(* Logix 5000 project; controller P3 vendor 1 type 14 code 92 rev 20.55; software revision 20.01 *)

TASK MainTask (continuous, watchdog 500 ms) : MainProgram

MODULES
   Local : vendor 1 type 14 code 92 (ICP 0, rev 20.55)
      P3_EN2T_PCN : 1756-EN2T (ICP 1, Ethernet 192.168.1.30, rev 10.1)
         P2 : 1756-EN2T (Ethernet 192.168.1.20, rev 10.1, Output RPI 10 ms)
            P2_CONTROLLER : vendor 1 type 14 code 92 (ICP 0, rev 20.1)
         P4 : 1756-EN2T (Ethernet 192.168.1.40, rev 10.1, Output RPI 10 ms)
            P4_CONTROLLER : vendor 1 type 14 code 92 (ICP 0, rev 20.1)
         P6 : 1756-EN2T (Ethernet 192.168.1.60, rev 10.1, Output RPI 10 ms)
            P6_CONTROLLER : vendor 1 type 14 code 92 (ICP 0, rev 20.1)
         EN2T_P1 : 1756-EN2T (Ethernet 192.168.1.10, rev 10.1, Output RPI 10 ms)
            P1_CONTROLLER : vendor 1 type 14 code 92 (ICP 0, rev 20.1)
         P5 : 1756-EN2T (Ethernet 192.168.1.50, rev 10.7, Output RPI 10 ms)
            P5_CONTROLLER : vendor 1 type 14 code 92 (ICP 0, rev 20.55)
      P3_EN2TR_RIO : vendor 1 type 12 code 200 (ICP 2, Ethernet 192.168.0.30, rev 10.1)
         RIO3 : 1794-AENTR (Ethernet 192.168.0.32, rev 1.1, Output RPI 20 ms)
            RIO3_DI : 1794-IB32 (Flex 0, rev 1.1, Input RPI 20 ms)
            RIO3_DO : vendor 1 type 7 code 35 (Flex 1, rev 1.1)
            RIO3_AI : 1794-IE12 (Flex 2, rev 1.1, Output RPI 78 ms)
         WRIO3 : vendor 309 type 12 code 1000 (Ethernet 192.168.0.35, rev 3.1, Output RPI 20 ms)
            WRIO3_AI : 1734-IE4C (PointIO 1, rev 3.1, Input RPI 80 ms)
END_MODULES

TYPE AIN_UDT :
STRUCT
   Pv : REAL;
   Heu : REAL;
   Leu : REAL;
   SAHH : REAL;
   SAH : REAL;
   SAL : REAL;
   SALL : REAL;
   AHH : BOOL;
   AH : BOOL;
   AL : BOOL;
   ALL : BOOL;
   Wifi_Enb : BOOL;
   Hty : BOOL;
   Sim : BOOL;
   Sim_PV : REAL;
END_STRUCT
END_TYPE

TYPE AUTOINP_UDT :
STRUCT
   ON : BOOL;
END_STRUCT
END_TYPE

TYPE ControllerLEDStatus :
STRUCT
   Off : BOOL;
   SolidGreen : BOOL;
   FlashingGreen : BOOL;
   SolidYellow : BOOL;
   FlashingYellow : BOOL;
   FlashingRed : BOOL;
   SolidRed : BOOL;
END_STRUCT
END_TYPE

TYPE Duty2_UDT :
STRUCT
   Selection : INT;
   Pump_Running : BOOL;
   Selected_Pmp_Not_Avl : BOOL;
   Both_Pmp_Not_Avl : BOOL;
END_STRUCT
END_TYPE

TYPE FaultRecord :
STRUCT
   timelow : DINT;
   timehigh : DINT;
   type : INT;
   code : INT;
   info : DINT[8];
END_STRUCT
END_TYPE

TYPE FIT_UDT :
STRUCT
   Pv : REAL;
   Heu : REAL;
   Leu : REAL;
   SAHH : REAL;
   SAH : REAL;
   SAL : REAL;
   SALL : REAL;
   Totaliser : REAL;
   AHH : BOOL;
   AH : BOOL;
   AL : BOOL;
   ALL : BOOL;
   Sim : BOOL;
   Sim_PV : REAL;
   Wifi_Enb : BOOL;
   Rst_Totaliser : BOOL;
   Hty : BOOL;
END_STRUCT
END_TYPE

TYPE Logix_Status_FP :
STRUCT
   ClearMinorFaults : DINT;
   Sts_MinorFaultEvents : DINT;
   Sts_MinorFaultBits : DINT;
   Sts_Redundant : DINT;
   Set_FaceplateAnimation : DINT;
   Val_ProductCode : DINT;
   MemoryTemp : INT[29];
   Val_raw_data : INT;
   Sts_IO_LED_raw : INT;
   Sts_ProductCode : INT;
   Val_Force_data_raw : INT;
   MemoryRequestData : SINT[12];
   Sts_Force_Installed : BOOL;
   Sts_Force_Enabled : BOOL;
   Sts_Faulted : BOOL;
   Sts_Run : BOOL;
   Sts_Program : BOOL;
   Sts_Minor_fault : BOOL;
   Sts_Major_fault : BOOL;
   Sts_KS_in_run : BOOL;
   Sts_KS_in_program : BOOL;
   Sts_KS_in_remote : BOOL;
   Sts_Changingmodes : BOOL;
   Sts_Test : BOOL;
   Sts_Ladder_Working : BOOL;
   Cmd_ClearFaultRecord : BOOL;
   Set_Controller_Description : STRING;
   UpdateDelayTimer : TIMER;
   Val_MajorFault : FaultRecord;
   Val_MFS : FaultRecord;
   Sts_IO_LED : ControllerLEDStatus;
   Sts_Battery_LED : ControllerLEDStatus;
   MemoryData : Memory_Data;
   TEST : DINT;
END_STRUCT
END_TYPE

TYPE Memory_Data :
STRUCT
   Free_Mem_IO : DINT;
   Free_Mem_DT : DINT;
   Free_Memory : DINT;
   Total_Mem_IO : DINT;
   Total_Mem_DT : DINT;
   Total_Memory : DINT;
   Biggest_IO_Mem_Size_Ava : DINT;
   Biggest_DT_Mem_Size_Ava : DINT;
END_STRUCT
END_TYPE

TYPE MV_UDT :
STRUCT
   Cmd : INT;
   Status : INT;
   Reset : BOOL;
   Auto : BOOL;
   FTO : BOOL;
   FTC : BOOL;
   Avl : BOOL;
END_STRUCT
END_TYPE

TYPE PLANT_AUTO_UDT :
STRUCT
   ON : BOOL;
   OFF : BOOL;
END_STRUCT
END_TYPE

TYPE PLANT_UDT :
STRUCT
   START : BOOL;
   STOP : BOOL;
END_STRUCT
END_TYPE

TYPE PMP_UDT :
STRUCT
   Cmd : INT;
   Status : INT;
   RunMin : REAL;
   Total_RunMin : REAL;
   RunHr : REAL;
   Total_RunHr : REAL;
   Remote : BOOL;
   Auto : BOOL;
   Fault : BOOL;
   Avl : BOOL;
   Permissive : DINT;
   Shutdown : DINT;
   SD : DINT;
   Reset : BOOL;
   Reset_RunHr : BOOL;
   FTR : BOOL;
   FTS : BOOL;
END_STRUCT
END_TYPE

TYPE PRECONDITION_UDT :
STRUCT
   PERMISSIVE1 : BOOL;
   PERMISSIVE2 : BOOL;
   PERMISSIVE3 : BOOL;
   PERMISSIVE4 : BOOL;
   PERMISSIVE5 : BOOL;
   SHUTDOWN1 : BOOL;
   SHUTDOWN2 : BOOL;
   SHUTDOWN3 : BOOL;
   SHUTDOWN4 : BOOL;
   SHUTDOWN5 : BOOL;
END_STRUCT
END_TYPE

TYPE RED_STAT :
STRUCT
   Redundancy_status_of_the_controller : INT;
   Redundancy_state_of_the_partner : INT;
END_STRUCT
END_TYPE

TYPE SWITCH_UDT :
STRUCT
   Alarm : BOOL;
   Delay : DINT;
END_STRUCT
END_TYPE

TYPE WIFI_UDT :
STRUCT
   PLC_WIFI : BOOL;
   RIO_WIFI : BOOL;
END_STRUCT
END_TYPE

ADD_ON_INSTRUCTION AIN_FBD   (* revision 1.0 *)
VAR_INPUT
   WRIO_Enb : BOOL; {visible}
   Raw_RIO : INT; {visible}
   Raw_WRIO : INT; {visible}
   L_Raw_RIO : INT; {visible}
   H_Raw_RIO : INT; {visible}
   L_Raw_WRIO : INT; {visible}
   H_Raw_WRIO : INT; {visible}
   HEU : INT; {visible}
   LEU : INT; {visible}
END_VAR
VAR_OUTPUT
   Hty : BOOL; {visible}
   Wifi_Enb : BOOL; {access Read Only, visible}
   AHH : BOOL; {visible}
   AH : BOOL; {access Read Only, visible}
   AL : BOOL; {access Read Only, visible}
   ALL : BOOL; {visible}
END_VAR
VAR_INPUT
   SAHH : REAL; {visible}
   SAH : REAL; {visible}
   SAL : REAL; {visible}
   SALL : REAL; {visible}
   Simulation : BOOL; {visible}
   RIO_Hty : BOOL; {visible}
   WRIO_Hty : BOOL; {visible}
END_VAR
VAR_IN_OUT
   Pv : REAL; {required}
   Sim_PV : REAL; {required}
   HMI : AIN_UDT; {required}
END_VAR
VAR
   SCALE : SCALE; {access None}
   ALM : ALARM; {access None}
   _Raw : INT; {access None}
   _L_Raw : INT; {access None}
   _H_Raw : INT; {access None}
   _Inst_Hty : BOOL; {access None}
END_VAR

ROUTINE Logic   (* structured text *)
   (*RIO and Wireless RIO Selection*)
   
   IF WRIO_Enb THEN
   	Wifi_Enb	:= 1;
   	_Raw		:= Raw_WRIO;
   	_H_Raw		:= H_Raw_WRIO;
   	_L_Raw		:= L_Raw_WRIO;
   	_Inst_Hty 	:= WRIO_Hty;
   ELSE
   	Wifi_Enb	:= 0;
   	_Raw		:= Raw_RIO;
   	_H_Raw		:= H_Raw_RIO;
   	_L_Raw		:= L_Raw_RIO;
   	_Inst_Hty 	:= RIO_Hty;
   END_IF;
   
   (*Calculation for PV*)
   IF Simulation THEN
   	Pv	:=Sim_PV;
   ELSE
   	SCALE.In		:=_Raw;
   	SCALE.InRawMax	:=_H_Raw;
   	SCALE.InRawMin	:=_L_Raw;
   	SCALE.InEUMax	:=HEU;
   	SCALE.InEUMin	:=LEU;
   	SCL(SCALE);
   
   	IF SCALE.Out<0 THEN
   		Pv	:= 0.0;
   	ELSE
   		Pv	:=SCALE.Out;
   	END_IF;
   
   	Sim_PV	:=Pv;
   
   END_IF;
   
   (*Alarms*)
   ALM.In			:=Pv;
   ALM.HHLimit		:=SAHH;
   ALM.HLimit		:=SAH;
   ALM.LLimit		:=SAL;
   ALM.LLLimit		:=SALL;
   ALM(ALM);
   
   AHH				:=ALM.HHAlarm;
   AH				:=ALM.HAlarm;
   AL				:=ALM.LAlarm;
   ALL				:=ALM.LLAlarm;
   
   Hty:= _Inst_Hty AND (_Raw > _L_Raw) AND (_Raw < _H_Raw)  ;
   
   
   
   
   
   
END_ROUTINE
END_ADD_ON_INSTRUCTION

ADD_ON_INSTRUCTION Duty2_FBD   (* revision 1.0 *)
VAR_INPUT
   AutoInp : BOOL; {visible}
   Selection : INT; {visible}
END_VAR
VAR_OUTPUT
   Start_Pmp1 : BOOL; {visible}
   Start_Pmp2 : BOOL; {visible}
END_VAR
VAR_IN_OUT
   PMP1 : PMP_UDT; {required}
   PMP2 : PMP_UDT; {required}
   HMI : Duty2_UDT; {required}
END_VAR

ROUTINE Logic   (* structured text *)
   IF PMP1.Status=2 OR PMP2.Status=2 THEN
   	HMI.Pump_Running := 1;
   ELSE
   	HMI.Pump_Running := 0;
   END_IF;
   
   IF AutoInp THEN
   	CASE Selection OF
   		(*PUMP 1 *)
   		1:
   			IF PMP1.Avl THEN
   				Start_Pmp1					:=1;
   				Start_Pmp2					:=0;
   				HMI.Selected_Pmp_Not_Avl	:=0;
   			ELSIF NOT PMP1.Avl AND PMP2.Avl THEN
   				Start_Pmp1					:=0;
   				Start_Pmp2					:=1;
   				HMI.Selected_Pmp_Not_Avl	:=1;
   			ELSIF NOT PMP1.Avl AND NOT PMP2.Avl	THEN
   				Start_Pmp1					:=0;
   				Start_Pmp2					:=0;
   				HMI.Both_Pmp_Not_Avl		:=1;
   			END_IF;
   
   		(*PUMP 2 *)
   		2:
   			IF PMP2.Avl THEN
   				Start_Pmp1					:=0;
   				Start_Pmp2					:=1;
   				HMI.Selected_Pmp_Not_Avl	:=0;
   			ELSIF NOT PMP2.Avl AND PMP1.Avl THEN
   				Start_Pmp1					:=1;
   				Start_Pmp2					:=0;
   				HMI.Selected_Pmp_Not_Avl	:=1;
   			ELSIF NOT PMP1.Avl AND NOT PMP2.Avl	THEN
   				Start_Pmp1					:=0;
   				Start_Pmp2					:=0;
   				HMI.Both_Pmp_Not_Avl		:=1;
   			END_IF;
   	END_CASE;
   ELSE
   	Start_Pmp1					:=0;
   	Start_Pmp2					:=0;
   END_IF;
   
   
END_ROUTINE
END_ADD_ON_INSTRUCTION

ADD_ON_INSTRUCTION FIT_FBD   (* revision 1.0 *)
VAR_INPUT
   WRIO_Enb : BOOL; {visible}
   Raw_RIO : INT; {visible}
   Raw_WRIO : INT; {visible}
   L_Raw_RIO : INT; {visible}
   H_Raw_RIO : INT; {visible}
   L_Raw_WRIO : INT; {visible}
   H_Raw_WRIO : INT; {visible}
   HEU : REAL; {visible}
   LEU : REAL; {visible}
END_VAR
VAR_OUTPUT
   Hty : BOOL; {visible}
   Wifi_Enb : BOOL; {visible}
   AHH : BOOL; {visible}
   AH : BOOL; {access Read Only, visible}
   AL : BOOL; {access Read Only, visible}
   ALL : BOOL; {visible}
END_VAR
VAR_INPUT
   SAHH : REAL; {visible}
   SAH : REAL; {visible}
   SAL : REAL; {visible}
   SALL : REAL; {visible}
   Simulation : BOOL; {visible}
   RIO_Hty : BOOL; {visible}
   WRIO_Hty : BOOL; {visible}
   Totaliser_Enb : BOOL; {visible}
   Rst_Totaliser : BOOL; {visible}
END_VAR
VAR_IN_OUT
   Totaliser : REAL; {required}
   Pv : REAL; {required}
   Sim_Pv : REAL; {required}
   HMI : FIT_UDT; {required}
END_VAR
VAR
   SCALE : SCALE; {access None}
   ALM : ALARM; {access None}
   TON : FBD_TIMER; {access None}
   _SEC_P : BOOL; {access None}
   _Inst_Hty : BOOL; {access None}
   _L_Raw : INT; {access None}
   _H_Raw : INT; {access None}
   _Raw : INT; {access None}
   R_TRIG : FBD_ONESHOT; {access None}
END_VAR

ROUTINE Logic   (* structured text *)
   (*RIO and Wireless RIO Selection*)
   
   IF WRIO_Enb THEN
   	Wifi_Enb	:= 1;
   	_Raw		:= Raw_WRIO;
   	_H_Raw		:= H_Raw_WRIO;
   	_L_Raw		:= L_Raw_WRIO;
   	_Inst_Hty 	:= WRIO_Hty;
   ELSE
   	Wifi_Enb	:= 0;
   	_Raw		:= Raw_RIO;
   	_H_Raw		:= H_Raw_RIO;
   	_L_Raw		:= L_Raw_RIO;
   	_Inst_Hty 	:= RIO_Hty;
   END_IF;
   
   (*Calculation for PV*)
   IF Simulation THEN
   	Pv	:= Sim_Pv   ;
   ELSE
   	SCALE.In		:=_Raw;
   	SCALE.InRawMax	:=_H_Raw;
   	SCALE.InRawMin	:=_L_Raw;
   	SCALE.InEUMax	:=HEU;
   	SCALE.InEUMin	:=LEU;
   	SCL(SCALE);
   	IF SCALE.Out>0 THEN
   		Pv	:=SCALE.Out;
   	ELSIF SCALE.Out<=0 THEN
   		Pv	:=0.0;
   	END_IF;
   
   	Sim_Pv	:=Pv;
   END_IF;
   
   (*Alarms*)
   ALM.In			:=Pv;
   ALM.HHLimit		:=SAHH;
   ALM.HLimit		:=SAH;
   ALM.LLimit		:=SAL;
   ALM.LLLimit		:=SALL;
   ALM(ALM);
   
   AHH				:=ALM.HHAlarm;
   AH				:=ALM.HAlarm;
   AL				:=ALM.LAlarm;
   ALL				:=ALM.LLAlarm;
   
   (*SECOND PULSE*)
   TON.PRE	:=1000;
   TON.TimerEnable	:=1;
   TONR(TON );
   R_TRIG.InputBit :=TON.DN ;
   OSRI( R_TRIG);
   _SEC_P  := R_TRIG.OutputBit;
   TON.Reset := _SEC_P;
   
   IF Totaliser_Enb THEN
   	IF _SEC_P THEN
   		HMI.Totaliser := HMI.Totaliser +  (ABS(Pv) / 3600 );
   	END_IF;
   END_IF;
   
   IF  Rst_Totaliser   THEN
   	HMI.Totaliser	:=0;
   END_IF;
   
   Hty:= _Inst_Hty AND (_Raw > _L_Raw) AND (_Raw < _H_Raw)  ;
   
   
   
   
   
   
END_ROUTINE
END_ADD_ON_INSTRUCTION

ADD_ON_INSTRUCTION MV_FBD   (* revision 1.0 *)
VAR_INPUT
   Auto : BOOL; {visible}
END_VAR
VAR_OUTPUT
   Cmd_Open : BOOL; {visible}
   Cmd_Close : BOOL; {visible}
   FTO : BOOL; {visible}
   FTC : BOOL; {access Read Only, visible}
END_VAR
VAR_INPUT
   AutoInp : BOOL; {visible}
   ZSO : BOOL; {visible}
   Open_TM : DINT; {visible}
   ZSC : BOOL; {visible}
   Close_TM : DINT; {visible}
END_VAR
VAR_IN_OUT
   Cmd : INT; {required}
   HMI : MV_UDT; {required}
END_VAR
VAR
   TON_Open_TM : FBD_TIMER; {access None}
   TON_Close_TM : FBD_TIMER; {access None}
END_VAR

ROUTINE Logic   (* structured text *)
   (*Fail to Close*)
   TON_Close_TM.PRE 			:= 	Close_TM*1000;
   TON_Close_TM.TimerEnable 	:=  Cmd_Close;
   TONR(TON_Close_TM);
   
   (*Fail to Open*)
   TON_Open_TM.PRE 			:= 	Open_TM*1000;
   TON_Open_TM.TimerEnable 	:= 	Cmd_Open;
   TONR(TON_Open_TM);
   
   IF ZSC THEN
   	HMI.Status	:=1;
   ELSIF ZSO THEN
   	HMI.Status	:=2;
   ELSE
   	HMI.Status	:=0;
   END_IF;
   
   HMI.Avl:= Auto AND NOT FTC AND NOT FTO;
   
   IF HMI.Reset THEN
   	(*IF NOT TON_Close_TM.DN AND ZSC THEN*)
   			FTC		:= 0;
   	(*END_IF;*)
   	(*IF NOT TON_Open_TM.DN AND ZSO THEN*)
   			FTO		:= 0;
   	(*END_IF;*)
   END_IF;
   
   IF  NOT Auto THEN
   	CASE HMI.Cmd OF
   		1:	(*CLOSE*)
   			Cmd_Close	:= 1;
   			Cmd_Open	:= 0;
   			IF TON_Close_TM.DN AND (NOT ZSC) THEN
   				FTC		:= 1;
   				FTO		:= 0;
   			END_IF;
   		2:	(*OPEN*)
   			IF FTO OR FTC    THEN
   				HMI.Cmd := 1;
   			END_IF;
   
   			IF NOT FTC AND NOT FTO THEN
   				Cmd_Close	:= 0;
   				Cmd_Open	:= 1;
   			END_IF;
   
   			IF TON_Open_TM.DN AND (NOT ZSO) THEN
   				FTC		:= 0;
   				FTO		:= 1;
   				HMI.Cmd := 1;
   			END_IF;
   	END_CASE;
   ELSE
   	(*Maintain Last status when switching from Auto to Manual*)
   	IF ZSO THEN
   		Cmd	:= 2;
   	END_IF;
   	IF ZSC THEN
   		Cmd	:= 1;
   	END_IF;
   
   	IF  AutoInp AND (NOT FTC AND NOT FTO) THEN
   		Cmd_Close	:= 0;
   		Cmd_Open	:= 1;
   		IF TON_Open_TM.DN AND (NOT ZSO) THEN
   			FTC		:= 0;
   			FTO		:= 1;
   		END_IF;
   	ELSE
   		Cmd_Close	:= 1;
   		Cmd_Open	:= 0;
   		IF TON_Close_TM.DN AND (NOT ZSC) THEN
   			FTC		:= 1;
   			FTO		:= 0;
   		END_IF;
   	END_IF;
   END_IF;
   
   
END_ROUTINE
END_ADD_ON_INSTRUCTION

ADD_ON_INSTRUCTION PMP_FBD   (* revision 1.0 *)
VAR_OUTPUT
   Cmd_Start : BOOL; {visible}
   Avl : BOOL; {visible}
   Fault : BOOL; {visible}
   FT_Stop : BOOL; {visible}
   FT_Start : BOOL; {visible}
   RunHr : REAL; {visible}
   Total_RunHr : REAL; {visible}
   SD : DINT; {access Read Only, visible}
END_VAR
VAR_INPUT
   Auto : BOOL; {visible}
   AutoInp : BOOL; {visible}
   Remote : BOOL; {visible}
   Run : BOOL; {visible}
   Trip : BOOL; {visible}
   Start_TM : DINT; {visible}
   Stop_TM : DINT; {visible}
   Rst : BOOL; {visible}
   Rst_RunHr : BOOL; {visible}
   Permissive : DINT; {visible}
   Shutdown : DINT; {visible}
END_VAR
VAR_IN_OUT
   RunMin : REAL; {required}
   Total_RunMin : REAL; {required}
   Cmd : INT; {required}
   HMI : PMP_UDT; {required}
END_VAR
VAR
   TON_Start_TM : FBD_TIMER; {access None}
   TON_Stop_TM : FBD_TIMER; {access None}
   _Min_P : BOOL; {access None}
   TON_Min : FBD_TIMER; {access None}
   R_TRIG_SEC : FBD_ONESHOT; {access None}
END_VAR

ROUTINE Logic   (* structured text *)
   (*Fail to Start*)
   TON_Start_TM.PRE 			:= 	Start_TM*1000;
   TON_Start_TM.TimerEnable 	:=  Cmd_Start;
   TONR(TON_Start_TM);
   
   (*Fail to Stop*)
   TON_Stop_TM.PRE 			:= 	Stop_TM*1000;
   TON_Stop_TM.TimerEnable 	:=  NOT Cmd_Start;
   TONR(TON_Stop_TM);
   
   IF (NOT Run) THEN
   	HMI.Status	:=1;
   ELSE
   	HMI.Status	:=2;
   END_IF;
   
   IF Fault THEN
   	HMI.Fault:= 1;
   ELSE
   	HMI.Fault:= 0;
   END_IF;
   
   IF HMI.Reset THEN
   	IF NOT TON_Stop_TM.DN THEN
   			FT_Stop		:= 0;
   	END_IF;
   	IF NOT TON_Start_TM.DN THEN
   			FT_Start	:= 0;
   	END_IF;
   
   	SD :=0;
   
   END_IF;
   
   Fault		:=Trip OR SD<>0;
   HMI.Remote	:=Remote;
   Avl:= Auto AND Remote AND NOT Fault AND NOT FT_Start AND NOT FT_Stop AND SD=0 ;
   
   IF Remote THEN
   	IF  NOT Auto THEN
   		CASE HMI.Cmd OF
   			1:	(*Stop*)
   				Cmd_Start	:=0;
   				IF TON_Stop_TM.DN AND Run THEN
   					FT_Start	:= 0;
   					FT_Stop		:= 1;
   				END_IF;
   			2:	(*OPEN*)
   				IF NOT Fault AND NOT FT_Start AND NOT FT_Stop AND (Permissive=-1) AND HMI.SD=0 THEN
   					Cmd_Start	:= 1;
   				ELSIF Cmd_Start AND (HMI.SD<>0) OR Fault THEN
   					SD				:= HMI.SD;
   					Cmd_Start		:= 0;
   					HMI.Cmd 		:= 1;
   				ELSIF (Permissive<>-1) THEN
   					HMI.Cmd 		:= 1;
   				END_IF;
   
   				IF TON_Start_TM.DN AND NOT Run THEN
   					FT_Start	:= 1;
   					FT_Stop		:= 0;
   					Cmd_Start	:= 0;
   					HMI.Cmd 	:= 1;
   				END_IF;
   		END_CASE;
   	ELSE
   		IF Run THEN
   			Cmd	:= 2;
   		END_IF;
   		IF (NOT Run) OR Fault OR FT_Start OR FT_Stop THEN
   			Cmd	:= 1;
   		END_IF;
   
   		IF  AutoInp  THEN
   			IF NOT Fault AND NOT FT_Start AND NOT FT_Stop AND (Permissive=-1) AND HMI.SD=0  THEN
   				Cmd_Start	:=1;
   			ELSIF ( Cmd_Start AND (HMI.SD<>0)) OR Fault THEN
   				SD			:= HMI.SD;
   				Cmd_Start	:=0;
   			END_IF;
   
   			IF TON_Start_TM.DN AND NOT Run THEN
   				FT_Start	:= 1;
   				FT_Stop		:= 0;
   				Cmd_Start	:= 0;
   				HMI.Cmd 	:= 1;
   			END_IF;
   		ELSE
   			Cmd_Start	:=0;
   			IF TON_Stop_TM.DN AND Run THEN
   				FT_Start	:= 0;
   				FT_Stop		:= 1;
   
   			END_IF;
   		END_IF;
   	END_IF;
   
   ELSE (*Local*)
   	Cmd_Start	:=0;
   	Cmd	:= 1;
   
   	FT_Start	:= 0;
   	FT_Stop		:= 0;
   
   
   
   
   	(*	IF Run THEN
   			Cmd	:= 2;
   		END_IF;
   		IF (NOT Run) OR Fault OR FT_Start OR FT_Stop THEN
   			Cmd	:= 1;
   		END_IF;
   		*)
   END_IF;
   
   (*1 MIN PULSE*)
   TON_Min.PRE	:=60000;
   TON_Min.TimerEnable	:=1;
   TONR(TON_Min );
   R_TRIG_SEC.InputBit :=TON_Min.DN ;
   OSRI( R_TRIG_SEC);
   _Min_P  := R_TRIG_SEC.OutputBit;
   TON_Min.Reset 	:= _Min_P;
   
   IF Run THEN
   	IF _Min_P THEN
   		RunMin 			:=RunMin + 1.0;
   		Total_RunMin	:=Total_RunMin + 1.0;
   	END_IF;
   END_IF;
   
   RunHr 				:=RunMin/60.0;
   Total_RunHr			:=Total_RunMin/60.0;
   
   IF  Rst_RunHr THEN
   	RunMin	:=0;
   END_IF;
   
   
   
END_ROUTINE
END_ADD_ON_INSTRUCTION

ADD_ON_INSTRUCTION SWITCH_FBD   (* revision 1.0 *)
VAR_INPUT
   Alarm : BOOL; {visible}
   Delay : DINT; {required}
END_VAR
VAR_OUTPUT
   Status : BOOL; {access None, required}
END_VAR
VAR_IN_OUT
   HMI : SWITCH_UDT; {required}
END_VAR
VAR
   TON_Delay_Sec : FBD_TIMER; {access None}
END_VAR

ROUTINE Logic   (* structured text *)
   (*Delay for Alarm*)
   TON_Delay_Sec.PRE 			:= 	Delay*1000;
   TON_Delay_Sec.TimerEnable 	:=  Alarm;
   TONR(TON_Delay_Sec);
   
   Status := TON_Delay_Sec.DN ;
END_ROUTINE
END_ADD_ON_INSTRUCTION

VAR_GLOBAL   (* controller tags *)
   _FIT301_Tot_Enb : BOOL;
   _LAST_STATE : INT := 1;
   _MIN_P : BOOL;
   _MV301_AutoInp : BOOL;
   _MV302_AutoInp : BOOL;
   _MV303_AutoInp : BOOL;
   _MV304_AutoInp : BOOL;
   _NEXT : BOOL;
   _ON_ENTRY : BOOL;
   _P301_AutoInp : BOOL;
   _P302_AutoInp : BOOL;
   _P602_AutoInp : BOOL;
   _P_NAOCL_UF_DUTY_AutoInp : BOOL;
   _P_UF_FEED_DUTY_AutoInp : BOOL;
   _SEC_P : BOOL;
   _SEC_P_2 : BOOL;
   AI_DPIT_301_DPRESS : INT := 708;
   AI_DPIT_301_DPRESS_HTY : BOOL := 1;
   AI_FIT_301_FLOW : INT := -12;
   AI_FIT_301_FLOW_HTY : BOOL := 1;
   AI_LIT_301_LEVEL : INT := 20324;
   AI_LIT_301_LEVEL_HTY : BOOL := 1;
   AI_RIO3_SPARE_03 : INT;
   AI_RIO3_SPARE_03_HTY : BOOL := 1;
   AI_RIO3_SPARE_04 : INT := -7701;
   AI_RIO3_SPARE_04_HTY : BOOL := 1;
   AI_RIO3_SPARE_05 : INT := -7702;
   AI_RIO3_SPARE_05_HTY : BOOL := 1;
   AI_RIO3_SPARE_06 : INT := -7704;
   AI_RIO3_SPARE_06_HTY : BOOL := 1;
   AI_RIO3_SPARE_07 : INT := -7701;
   AI_RIO3_SPARE_07_HTY : BOOL := 1;
   AI_RIO3_SPARE_08 : INT := -7700;
   AI_RIO3_SPARE_08_HTY : BOOL := 1;
   AI_RIO3_SPARE_09 : INT := -7703;
   AI_RIO3_SPARE_09_HTY : BOOL := 1;
   AI_RIO3_SPARE_10 : INT := -7700;
   AI_RIO3_SPARE_10_HTY : BOOL := 1;
   AI_RIO3_SPARE_11 : INT := -7701;
   AI_RIO3_SPARE_11_HTY : BOOL := 1;
   DI_DPSH_301_HIGH : BOOL;
   DI_MV_301_ZSC : BOOL := 1;
   DI_MV_301_ZSO : BOOL;
   DI_MV_302_ZSC : BOOL := 1;
   DI_MV_302_ZSO : BOOL;
   DI_MV_303_ZSC : BOOL := 1;
   DI_MV_303_ZSO : BOOL;
   DI_MV_304_ZSC : BOOL := 1;
   DI_MV_304_ZSO : BOOL;
   DI_P_301_AUTO : BOOL := 1;
   DI_P_301_FAULT : BOOL;
   DI_P_301_RUN : BOOL;
   DI_P_302_AUTO : BOOL := 1;
   DI_P_302_FAULT : BOOL;
   DI_P_302_RUN : BOOL;
   DI_PSH_301_HIGH : BOOL;
   DI_RIO3_SPARE_18 : BOOL;
   DI_RIO3_SPARE_19 : BOOL;
   DI_RIO3_SPARE_20 : BOOL;
   DI_RIO3_SPARE_21 : BOOL;
   DI_RIO3_SPARE_22 : BOOL;
   DI_RIO3_SPARE_23 : BOOL;
   DI_RIO3_SPARE_24 : BOOL;
   DI_RIO3_SPARE_25 : BOOL;
   DI_RIO3_SPARE_26 : BOOL;
   DI_RIO3_SPARE_27 : BOOL;
   DI_RIO3_SPARE_28 : BOOL;
   DI_RIO3_SPARE_29 : BOOL;
   DI_RIO3_SPARE_30 : BOOL;
   DI_RIO3_SPARE_31 : BOOL;
   DI_WIFI_PLC_3 : BOOL;
   DI_WIFI_RIO_3 : BOOL;
   DO_MV_301_CLOSE : BOOL := 1;
   DO_MV_301_OPEN : BOOL;
   DO_MV_302_CLOSE : BOOL := 1;
   DO_MV_302_OPEN : BOOL;
   DO_MV_303_CLOSE : BOOL := 1;
   DO_MV_303_OPEN : BOOL;
   DO_MV_303_START : BOOL;
   DO_MV_304_CLOSE : BOOL := 1;
   DO_MV_304_OPEN : BOOL;
   DO_P_301_START : BOOL;
   DO_P_302_START : BOOL;
   DO_RIO2_SPARE_10 : BOOL;
   DO_RIO3_SPARE_10 : BOOL;
   DO_RIO3_SPARE_11 : BOOL;
   DO_RIO3_SPARE_12 : BOOL;
   DO_RIO3_SPARE_13 : BOOL;
   DO_RIO3_SPARE_14 : BOOL;
   DO_RIO3_SPARE_15 : BOOL;
   DPIT301_FB : AIN_FBD := (Raw_RIO := 708, Raw_WRIO := 3256, L_Raw_RIO := -30, H_Raw_RIO := 31208, L_Raw_WRIO := 3277, H_Raw_WRIO := 16383, HEU := 100, Hty := 1, AL := 1, ALL := 1, SAHH := 100.0, SAH := 40.0, SAL := 15.0, SALL := 10.0, RIO_Hty := 1, WRIO_Hty := 1);
   DPSH301_FB : SWITCH_FBD;
   ERROR_P3_Le : REAL;
   ERROR_P3_Ls : REAL := 0.08013916;
   FIT301_FB : FIT_FBD := (Raw_RIO := -12, Raw_WRIO := 3260, L_Raw_RIO := -15, H_Raw_RIO := 31208, L_Raw_WRIO := 3277, H_Raw_WRIO := 16383, HEU := 4.0, Hty := 1, SAHH := 3.5, SAH := 3.0, RIO_Hty := 1, WRIO_Hty := 1);
   HMI_BACKWASH_SEC : INT;
   HMI_BACKWASH_SEC_SP : INT := 30;
   HMI_BW_CNT : INT := 83;
   HMI_CIP_CLEANING_SEC : INT;
   HMI_CIP_CLEANING_SEC_SP : INT := 30;
   HMI_DPIT301 : AIN_UDT := (Pv := 2.362507, SAHH := 100.0, SAH := 40.0, SAL := 15.0, SALL := 10.0, AL := 1, ALL := 1, Hty := 1, Sim_PV := 2.362507);
   HMI_DPS301 : SWITCH_UDT;
   HMI_DPSH301 : SWITCH_UDT;
   HMI_DRAIN_SEC : INT;
   HMI_DRAIN_SEC_SP : INT := 45;
   HMI_FIT201 : FIT_UDT := (SAHH := 3.5, SAH := 2.0, Totaliser := 35.307026, AL := 1, ALL := 1);
   HMI_FIT301 : FIT_UDT := (Pv := 0.00038433203, SAHH := 3.5, SAH := 3.0, Totaliser := 202.71819, Sim_PV := 0.00038433203, Hty := 1);
   HMI_LIT101 : AIN_UDT := (Pv := 868.4317, SAHH := 1100.0, SAH := 800.0, SAL := 500.0, SALL := 250.0, AH := 1, Hty := 1, Sim := 1, Sim_PV := 868.4317);
   HMI_LIT301 : AIN_UDT := (Pv := 814.2143, SAHH := 1200.0, SAH := 1000.0, SAL := 800.0, SALL := 250.0, Hty := 1, Sim_PV := 814.2143);
   HMI_LIT401 : AIN_UDT := (Pv := 799.21814, SAHH := 1200.0, SAH := 800.0, SAL := 800.0, SALL := 250.0, AL := 1, Hty := 1, Sim_PV := 799.21814);
   HMI_MV201 : MV_UDT := (Cmd := 1, Status := 1, Auto := 1, Avl := 1);
   HMI_MV301 : MV_UDT := (Cmd := 1, Status := 1, Reset := 1, Auto := 1, Avl := 1);
   HMI_MV302 : MV_UDT := (Cmd := 1, Status := 1, Reset := 1, Auto := 1, Avl := 1);
   HMI_MV303 : MV_UDT := (Cmd := 1, Status := 1, Reset := 1, Auto := 1, Avl := 1);
   HMI_MV304 : MV_UDT := (Cmd := 1, Status := 1, Reset := 1, Auto := 1, Avl := 1);
   HMI_P101 : PMP_UDT := (Cmd := 1, Status := 1, RunMin := 1558.0, Total_RunMin := 1558.0, RunHr := 25.966667, Total_RunHr := 25.966667, Remote := 1, Permissive := -3, Reset := 1);
   HMI_P301 : PMP_UDT := (Cmd := 1, Status := 1, RunMin := 5986.0, Total_RunMin := 5986.0, RunHr := 99.76667, Total_RunHr := 99.76667, Remote := 1, Auto := 1, Avl := 1, Permissive := -5, Reset := 1);
   HMI_P301_MSG : PRECONDITION_UDT := (PERMISSIVE1 := 1, PERMISSIVE2 := 1);
   HMI_P302 : PMP_UDT := (Cmd := 1, Status := 1, RunMin := 706.0, Total_RunMin := 706.0, RunHr := 11.766666, Total_RunHr := 11.766666, Remote := 1, Auto := 1, Avl := 1, Permissive := -5, Reset := 1);
   HMI_P302_MSG : PRECONDITION_UDT := (PERMISSIVE1 := 1, PERMISSIVE2 := 1);
   HMI_P3_PERMISSIVE : AUTOINP_UDT := (ON := 1);
   HMI_P3_SHUTDOWN : BOOL;
   HMI_P3_STATE : INT := 1;
   HMI_P602 : PMP_UDT := (Cmd := 1, Status := 1, RunMin := 63.0, Total_RunMin := 63.0, RunHr := 1.05, Total_RunHr := 1.05, Remote := 1, Auto := 1, Avl := 1, Permissive := -1, Reset := 1);
   HMI_P_NAOCL_UF_DUTY : Duty2_UDT := (Selection := 2);
   HMI_P_UF_FEED_DUTY : Duty2_UDT := (Selection := 1, Both_Pmp_Not_Avl := 1);
   HMI_PLANT : PLANT_UDT;
   HMI_PLANT_AUTO : PLANT_AUTO_UDT;
   HMI_PLANT_PERMISSIVE : BOOL;
   HMI_PLANT_RESET : PLANT_AUTO_UDT;
   HMI_PSH301 : SWITCH_UDT;
   HMI_START_PLANT : BOOL;
   HMI_STOP_PLANT : BOOL;
   HMI_TMP_HIGH : BOOL;
   HMI_UF_FILTRATION_MIN : INT;
   HMI_UF_FILTRATION_MIN_SP : INT := 30;
   HMI_UF_REFILL_SEC : INT;
   HMI_UF_REFILL_SEC_SP : INT := 30;
   HMI_WIFI : WIFI_UDT;
   Le_Error_Occured : BOOL;
   LIT301_FB : AIN_FBD := (Raw_RIO := 20331, Raw_WRIO := 9279, H_Raw_RIO := 31208, L_Raw_WRIO := 3277, H_Raw_WRIO := 16383, HEU := 1250, Hty := 1, SAHH := 1200.0, SAH := 1000.0, SAL := 800.0, SALL := 250.0, RIO_Hty := 1, WRIO_Hty := 1);
   LIT_301_Le_PRV : REAL := 852.30554;
   LIT_301_Ls_PRV : REAL := 814.0541;
   LIT_301_MODEL_Le : REAL := 948.25653;
   LIT_301_MODEL_Ls : REAL := 813.97394;
   LIT_301_VALID : BOOL;
   LIT_ALM : ALARM := (In := 948.25653, HHLimit := 1100.0, HLimit := 800.0, LLimit := 500.0, LLLimit := 250.0, HAlarm := 1);
   LIT_DELTA : REAL := 363.2074;
   LIT_SEC : DINT := 277;
   LIT_SEC_SP : DINT := 5;
   LIT_STATE : INT := 2;
   Logix_Status : Logix_Status_FP := (Set_FaceplateAnimation := 90, Val_ProductCode := 92, MemoryTemp[0] := 5, MemoryTemp[1] := 1, MemoryTemp[3] := 28010, MemoryTemp[4] := 3, MemoryTemp[5] := -138, MemoryTemp[6] := 6, MemoryTemp[9] := 2, MemoryTemp[11] := -4608, MemoryTemp[12] := 3, MemoryTemp[14] := 8, MemoryTemp[17] := 5, MemoryTemp[21] := 6, MemoryTemp[23] := 25968, MemoryTemp[24] := 3, MemoryTemp[25] := 7, MemoryTemp[27] := -138, MemoryTemp[28] := 6, Val_raw_data := 12384, Sts_IO_LED_raw := 2, Sts_ProductCode := 92, MemoryRequestData[0] := 5, MemoryRequestData[2] := 1, MemoryRequestData[4] := 2, MemoryRequestData[6] := 5, MemoryRequestData[8] := 6, MemoryRequestData[10] := 7, Sts_Run := 1, Sts_KS_in_remote := 1, Sts_Ladder_Working := 1, Set_Controller_Description := 'P3: Ultra-Filtration System', UpdateDelayTimer.PRE := 1000, UpdateDelayTimer.ACC := 767, UpdateDelayTimer.EN := 1, UpdateDelayTimer.TT := 1, Val_MFS.timelow := 71751885, Val_MFS.timehigh := 206334, Val_MFS.type := 3, Val_MFS.code := 20, Val_MFS.info[1] := 1, Sts_IO_LED.FlashingGreen := 1, Sts_Battery_LED.Off := 1, MemoryData.Free_Mem_IO := 898472, MemoryData.Free_Mem_DT := 1834456, MemoryData.Total_Mem_IO := 1030144, MemoryData.Total_Mem_DT := 2097152, MemoryData.Biggest_IO_Mem_Size_Ava := 890304, MemoryData.Biggest_DT_Mem_Size_Ava := 1834456);
   Ls_Error_Occured : BOOL;
   Memory_Message : MESSAGE;
        MessageParameters(ServiceCode := 16#0003, LocalElement := Logix_Status.MemoryRequestData[0], DestinationTag := Logix_Status.MemoryTemp[0], ...)
   MIN_TEST : DINT := 268293;
   MV301_FB : MV_FBD := (Auto := 1, Cmd_Close := 1, Open_TM := 10, ZSC := 1, Close_TM := 10);
   MV302_FB : MV_FBD := (Auto := 1, Cmd_Close := 1, Open_TM := 10, ZSC := 1, Close_TM := 10);
   MV303_FB : MV_FBD := (Auto := 1, Cmd_Close := 1, Open_TM := 10, ZSC := 1, Close_TM := 10);
   MV304_FB : MV_FBD := (Auto := 1, Cmd_Close := 1, Open_TM := 10, ZSC := 1, Close_TM := 10);
   P1_LIT101_MSG : MESSAGE;
        MessageParameters(ServiceCode := 16#004c, LocalElement := HMI_LIT101, ...)
   P1_P101_MSG : MESSAGE;
        MessageParameters(ServiceCode := 16#004c, LocalElement := HMI_P101, ...)
   P1_P101_MSG2 : MESSAGE;
        MessageParameters(ServiceCode := 16#004c, LocalElement := HMI_P101, ...)
   P2_FIT201_MSG : MESSAGE;
        MessageParameters(ServiceCode := 16#004c, LocalElement := HMI_FIT201, ...)
   P2_MV201_MSG : MESSAGE;
        MessageParameters(ServiceCode := 16#004c, LocalElement := HMI_MV201, ...)
   P2_P2078_AUTOINP : AUTOINP_UDT;
   P2_P2078_CMD_MSG : MESSAGE;
        MessageParameters(ServiceCode := 16#004d, LocalElement := P2_P2078_AUTOINP, ...)
   P2_P2078_MSG : MESSAGE;
        MessageParameters(ServiceCode := 16#004c, LocalElement := HMI_P_NAOCL_UF_DUTY, ...)
   P301_FB : PMP_FBD := (Avl := 1, RunHr := 99.76667, Total_RunHr := 99.76667, Auto := 1, Remote := 1, Start_TM := 3, Stop_TM := 3, Rst := 1, Permissive := -5);
   P302_FB : PMP_FBD := (Avl := 1, RunHr := 11.766666, Total_RunHr := 11.766666, Auto := 1, Remote := 1, Start_TM := 3, Stop_TM := 3, Rst := 1, Permissive := -5);
   P4_LIT401_MSG : MESSAGE;
        MessageParameters(ServiceCode := 16#004c, LocalElement := HMI_LIT401, ...)
   P6_P602_AUTOINP : AUTOINP_UDT;
   P6_P602_CMD_MSG : MESSAGE;
        MessageParameters(ServiceCode := 16#004d, LocalElement := P6_P602_AUTOINP, ...)
   P6_P602_MSG : MESSAGE;
        MessageParameters(ServiceCode := 16#004c, LocalElement := HMI_P602, ...)
   P6_P_BW_MSG : MESSAGE;
        MessageParameters(ServiceCode := 16#004c, LocalElement := HMI_P602, ...)
   P_UF_FEED_DUTY_FB : Duty2_FBD := (Selection := 1);
   PLANT_CRITICAL_SD : AUTOINP_UDT;
   PSH301_FB : SWITCH_FBD;
   R_TRIG : FBD_ONESHOT;
   R_TRIG1 : FBD_ONESHOT;
   R_TRIG_BW : FBD_ONESHOT;
   REDUNDANT_STATUS : RED_STAT := (Redundancy_status_of_the_controller := 2, Redundancy_state_of_the_partner := 8);
   RTRIG_MIN : FBD_ONESHOT;
   SEC_TEST : INT := 40;
   TON : FBD_TIMER := (TimerEnable := 1, PRE := 1000, ACC := 695, EN := 1, TT := 1);
   TON1 : FBD_TIMER := (TimerEnable := 1, PRE := 1000, ACC := 850, EN := 1, TT := 1);
   TON_FIT301_P1_TM : FBD_TIMER := (PRE := 6000);
   TON_FIT301_P2_TM : FBD_TIMER := (PRE := 6000);
   TON_FIT302_TM : FBD_TIMER := (PRE := 6000);
   TON_MIN : FBD_TIMER := (TimerEnable := 1, PRE := 60000, ACC := 6041, EN := 1, TT := 1);
   W_AI_DPIT_301_DPRESS : INT := 3256;
   W_AI_DPIT_301_DPRESS_HTY : BOOL := 1;
   W_AI_FIT_301_FLOW : INT := 3260;
   W_AI_FIT_301_FLOW_HTY : BOOL := 1;
   W_AI_LIT_301_LEVEL : INT := 9279;
   W_AI_LIT_301_LEVEL_HTY : BOOL := 1;
   W_AI_RIO3_SPARE_03 : INT := -4;
   W_AI_RIO3_SPARE_03_HTY : BOOL;
END_VAR

PROGRAM MainProgram   (* main routine MainRoutine *)
VAR
   _P_UF_FEED_DUTY_SR : DOMINANT_SET := (Out := 1);
   _SEC_P3 : BOOL;
   ATTACK : BOOL := 1;
   avg : REAL := 0.1602234;
   count : DINT := 3;
   Error_list : REAL[10] := ([0] := 0.08013916, [1] := 0.28045654, [2] := 6.1035156e-05, [3] := 0.039978027, [4] := 0.3204956, [5] := 0.20019531, [6] := 6.1035156e-05, [7] := 0.28033447, [8] := 0.36053467, [9] := 0.039978027);
   first : BOOL := 1;
   TEMP_P3 : REAL;
END_VAR

ROUTINE IO   (* structured text *)
   (*DIGITAL INPUTS*)
   DI_WIFI_PLC_3	:=RIO3:0:I.Data.0;
   DI_WIFI_RIO_3	:=RIO3:0:I.Data.1;
   DI_P_301_AUTO	:=RIO3:0:I.Data.2;
   DI_P_301_RUN	:=RIO3:0:I.Data.3;
   DI_P_301_FAULT	:=RIO3:0:I.Data.4;
   DI_P_302_AUTO	:=RIO3:0:I.Data.5;
   DI_P_302_RUN	:=RIO3:0:I.Data.6;
   DI_P_302_FAULT	:=RIO3:0:I.Data.7;
   DI_MV_301_ZSO	:=RIO3:0:I.Data.8;
   DI_MV_301_ZSC	:=RIO3:0:I.Data.9;
   DI_MV_302_ZSO	:=RIO3:0:I.Data.10;
   DI_MV_302_ZSC	:=RIO3:0:I.Data.11;
   DI_MV_303_ZSO	:=RIO3:0:I.Data.12;
   DI_MV_303_ZSC	:=RIO3:0:I.Data.13;
   DI_MV_304_ZSO	:=RIO3:0:I.Data.14;
   DI_MV_304_ZSC	:=RIO3:0:I.Data.15;
   DI_PSH_301_HIGH	:=RIO3:0:I.Data.16;
   DI_DPSH_301_HIGH:=RIO3:0:I.Data.17;
   DI_RIO3_SPARE_18:=RIO3:0:I.Data.18;
   DI_RIO3_SPARE_19:=RIO3:0:I.Data.19;
   DI_RIO3_SPARE_20:=RIO3:0:I.Data.20;
   DI_RIO3_SPARE_21:=RIO3:0:I.Data.21;
   DI_RIO3_SPARE_22:=RIO3:0:I.Data.22;
   DI_RIO3_SPARE_23:=RIO3:0:I.Data.23;
   DI_RIO3_SPARE_24:=RIO3:0:I.Data.24;
   DI_RIO3_SPARE_25:=RIO3:0:I.Data.25;
   DI_RIO3_SPARE_26:=RIO3:0:I.Data.26;
   DI_RIO3_SPARE_27:=RIO3:0:I.Data.27;
   DI_RIO3_SPARE_28:=RIO3:0:I.Data.28;
   DI_RIO3_SPARE_29:=RIO3:0:I.Data.29;
   DI_RIO3_SPARE_30:=RIO3:0:I.Data.30;
   DI_RIO3_SPARE_31:=RIO3:0:I.Data.31;
   
   (*DIGITAL OUTPUTS*)
   RIO3:1:O.0	:=DO_P_301_START;
   RIO3:1:O.1	:=DO_P_302_START;
   RIO3:1:O.2	:=DO_MV_301_OPEN;
   RIO3:1:O.3	:=DO_MV_301_CLOSE;
   RIO3:1:O.4	:=DO_MV_302_OPEN;
   RIO3:1:O.5	:=DO_MV_302_CLOSE;
   RIO3:1:O.6	:=DO_MV_303_OPEN;
   RIO3:1:O.7	:=DO_MV_303_CLOSE;
   RIO3:1:O.8	:=DO_MV_304_OPEN;
   RIO3:1:O.9	:=DO_MV_304_CLOSE;
   RIO3:1:O.10	:=DO_RIO3_SPARE_10;
   RIO3:1:O.11	:=DO_RIO3_SPARE_11;
   RIO3:1:O.12	:=DO_RIO3_SPARE_12;
   RIO3:1:O.13	:=DO_RIO3_SPARE_13;
   RIO3:1:O.14	:=DO_RIO3_SPARE_14;
   RIO3:1:O.15	:=DO_RIO3_SPARE_15;
   
   (*ANALOG INPUTS*)
   AI_LIT_301_LEVEL	:=RIO3:2:I.Ch0Data;
   AI_FIT_301_FLOW		:=RIO3:2:I.Ch1Data;
   AI_DPIT_301_DPRESS	:=RIO3:2:I.Ch2Data;
   AI_RIO3_SPARE_04	:=RIO3:2:I.Ch4Data;
   AI_RIO3_SPARE_05	:=RIO3:2:I.Ch5Data;
   AI_RIO3_SPARE_06	:=RIO3:2:I.Ch6Data;
   AI_RIO3_SPARE_07	:=RIO3:2:I.Ch7Data;
   AI_RIO3_SPARE_08	:=RIO3:2:I.Ch8Data;
   AI_RIO3_SPARE_09	:=RIO3:2:I.Ch9Data;
   AI_RIO3_SPARE_10	:=RIO3:2:I.Ch10Data;
   AI_RIO3_SPARE_11	:=RIO3:2:I.Ch11Data;
   
   AI_LIT_301_LEVEL_HTY	:=(NOT RIO3:2:I.GeneralFault);
   AI_FIT_301_FLOW_HTY		:=(NOT RIO3:2:I.GeneralFault);
   AI_DPIT_301_DPRESS_HTY	:=(NOT RIO3:2:I.GeneralFault);
   AI_RIO3_SPARE_03_HTY	:=(NOT RIO3:2:I.GeneralFault);
   AI_RIO3_SPARE_04_HTY	:=(NOT RIO3:2:I.GeneralFault);
   AI_RIO3_SPARE_05_HTY	:=(NOT RIO3:2:I.GeneralFault);
   AI_RIO3_SPARE_06_HTY	:=(NOT RIO3:2:I.GeneralFault);
   AI_RIO3_SPARE_07_HTY	:=(NOT RIO3:2:I.GeneralFault);
   AI_RIO3_SPARE_08_HTY	:=(NOT RIO3:2:I.GeneralFault);
   AI_RIO3_SPARE_09_HTY	:=(NOT RIO3:2:I.GeneralFault);
   AI_RIO3_SPARE_10_HTY	:=(NOT RIO3:2:I.GeneralFault);
   AI_RIO3_SPARE_11_HTY	:=(NOT RIO3:2:I.GeneralFault);
   
   (*WIRELESS ANALOG INPUTS*)
   W_AI_LIT_301_LEVEL		:=WRIO3:1:I.Ch0Data;
   W_AI_FIT_301_FLOW		:=WRIO3:1:I.Ch1Data;
   W_AI_DPIT_301_DPRESS	:=WRIO3:1:I.Ch2Data;
   W_AI_RIO3_SPARE_03		:=WRIO3:1:I.Ch3Data;
   
   W_AI_LIT_301_LEVEL_HTY		:=(NOT WRIO3:1:I.Ch0Fault);
   W_AI_FIT_301_FLOW_HTY		:=(NOT WRIO3:1:I.Ch1Fault);
   W_AI_DPIT_301_DPRESS_HTY	:=(NOT WRIO3:1:I.Ch2Fault);
   W_AI_RIO3_SPARE_03_HTY		:=(NOT WRIO3:1:I.Ch3Fault);
   
   (*Wireless Selction*)
   HMI_WIFI.PLC_WIFI		:= DI_WIFI_PLC_3;
   HMI_WIFI.RIO_WIFI		:= DI_WIFI_RIO_3;
   
END_ROUTINE

ROUTINE Logix_Status   (* ladder *)
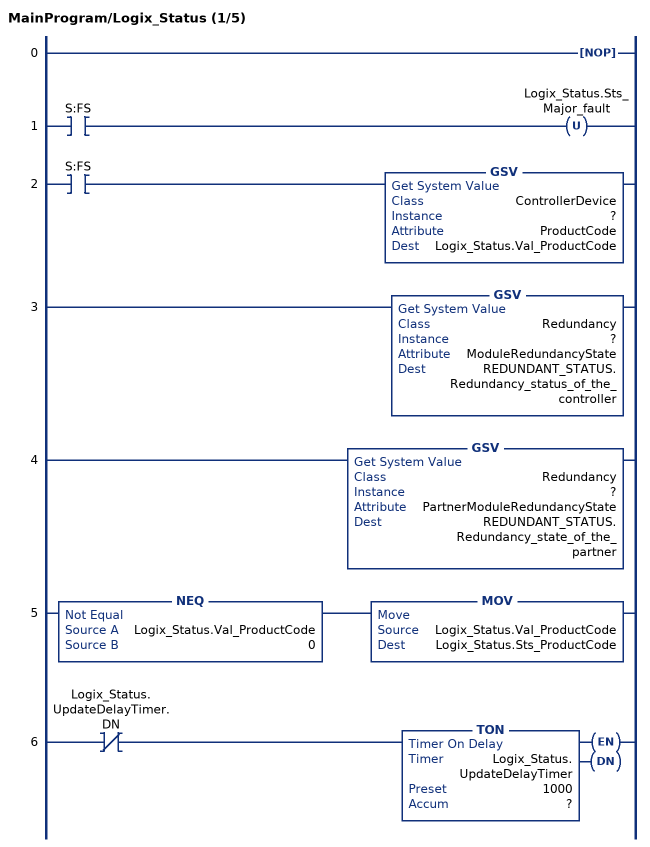
   0: NOP();
   1: XIC(S:FS)OTU(Logix_Status.Sts_Major_fault);
   2: XIC(S:FS)GSV(ControllerDevice,?,ProductCode,Logix_Status.Val_ProductCode);
   3: GSV(Redundancy,?,ModuleRedundancyState,REDUNDANT_STATUS.Redundancy_status_of_the_controller);
   4: GSV(Redundancy,?,PartnerModuleRedundancyState,REDUNDANT_STATUS.Redundancy_state_of_the_partner);
   5: NEQ(Logix_Status.Val_ProductCode,0)MOV(Logix_Status.Val_ProductCode,Logix_Status.Sts_ProductCode);
   6: XIO(Logix_Status.UpdateDelayTimer.DN)TON(Logix_Status.UpdateDelayTimer,?,?);
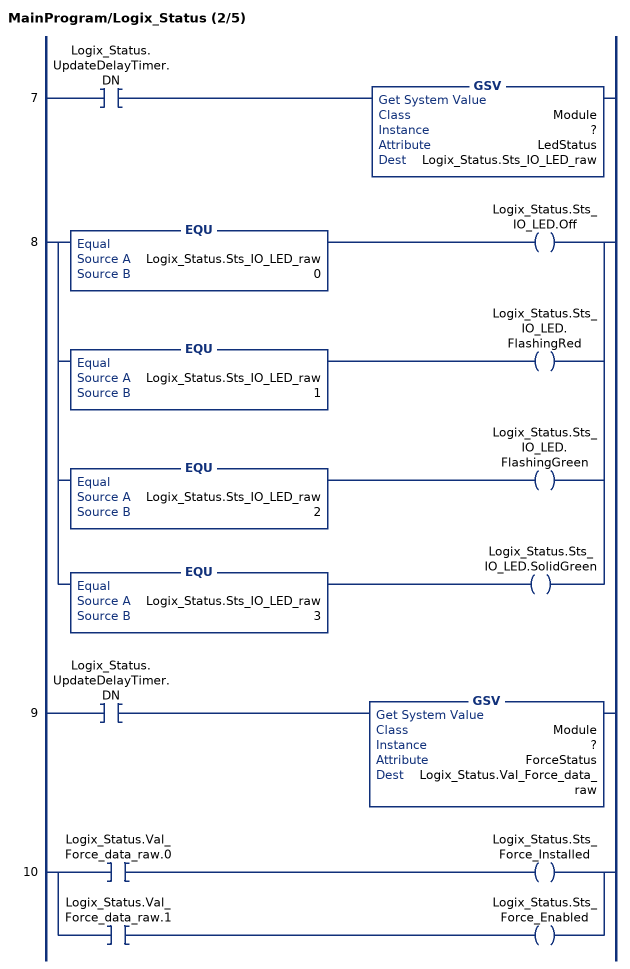
   7: XIC(Logix_Status.UpdateDelayTimer.DN)GSV(Module,?,LedStatus,Logix_Status.Sts_IO_LED_raw);
   8: [EQU(Logix_Status.Sts_IO_LED_raw,0) OTE(Logix_Status.Sts_IO_LED.Off) ,EQU(Logix_Status.Sts_IO_LED_raw,1) OTE(Logix_Status.Sts_IO_LED.FlashingRed) ,EQU(Logix_Status.Sts_IO_LED_raw,2) OTE(Logix_Status.Sts_IO_LED.FlashingGreen) ,EQU(Logix_Status.Sts_IO_LED_raw,3) OTE(Logix_Status.Sts_IO_LED.SolidGreen) ];
   9: XIC(Logix_Status.UpdateDelayTimer.DN)GSV(Module,?,ForceStatus,Logix_Status.Val_Force_data_raw);
   10: [XIC(Logix_Status.Val_Force_data_raw.0) OTE(Logix_Status.Sts_Force_Installed) ,XIC(Logix_Status.Val_Force_data_raw.1) OTE(Logix_Status.Sts_Force_Enabled) ];
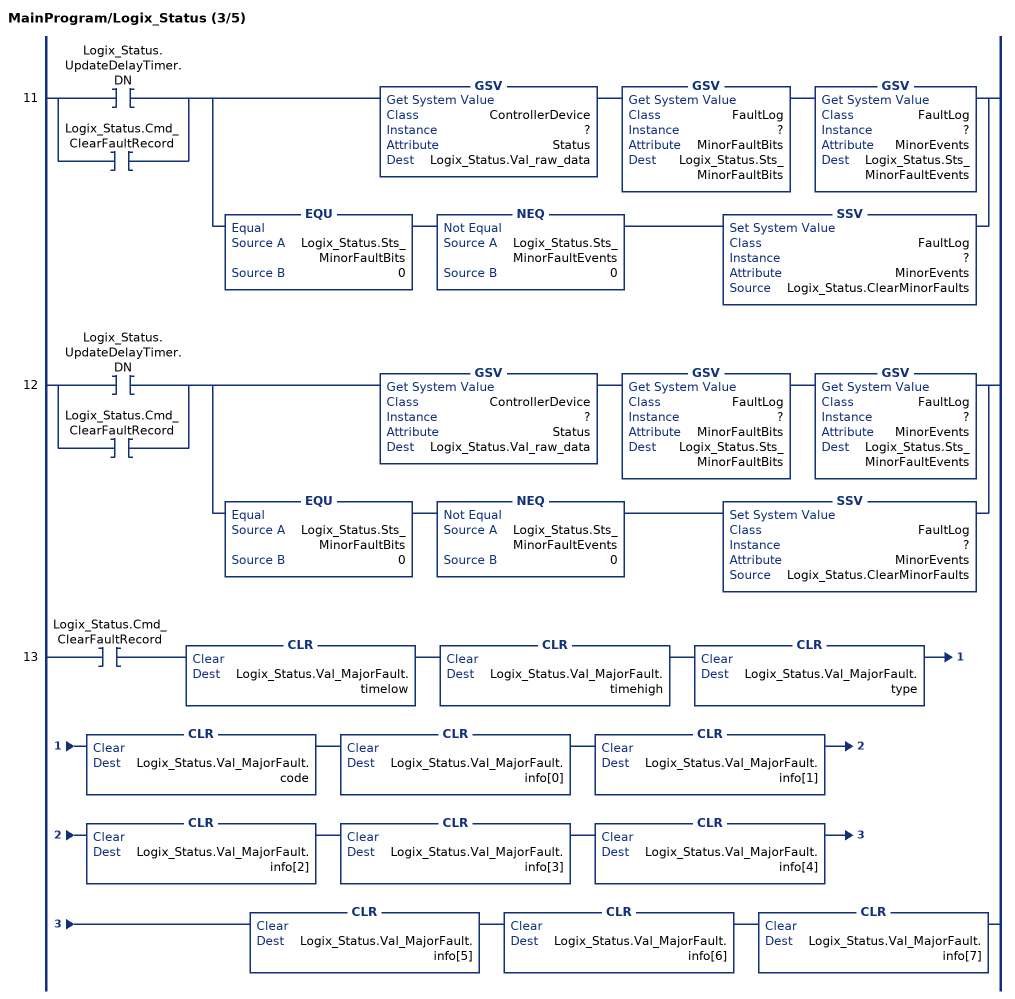
   11: [XIC(Logix_Status.UpdateDelayTimer.DN) ,XIC(Logix_Status.Cmd_ClearFaultRecord) ][GSV(ControllerDevice,?,Status,Logix_Status.Val_raw_data) GSV(FaultLog,?,MinorFaultBits,Logix_Status.Sts_MinorFaultBits) GSV(FaultLog,?,MinorEvents,Logix_Status.Sts_MinorFaultEvents) ,EQU(Logix_Status.Sts_MinorFaultBits,0) NEQ(Logix_Status.Sts_MinorFaultEvents,0) SSV(FaultLog,?,MinorEvents,Logix_Status.ClearMinorFaults) ];
   12: [XIC(Logix_Status.UpdateDelayTimer.DN) ,XIC(Logix_Status.Cmd_ClearFaultRecord) ][GSV(ControllerDevice,?,Status,Logix_Status.Val_raw_data) GSV(FaultLog,?,MinorFaultBits,Logix_Status.Sts_MinorFaultBits) GSV(FaultLog,?,MinorEvents,Logix_Status.Sts_MinorFaultEvents) ,EQU(Logix_Status.Sts_MinorFaultBits,0) NEQ(Logix_Status.Sts_MinorFaultEvents,0) SSV(FaultLog,?,MinorEvents,Logix_Status.ClearMinorFaults) ];
   13: XIC(Logix_Status.Cmd_ClearFaultRecord)CLR(Logix_Status.Val_MajorFault.timelow)CLR(Logix_Status.Val_MajorFault.timehigh)CLR(Logix_Status.Val_MajorFault.type)CLR(Logix_Status.Val_MajorFault.code)CLR(Logix_Status.Val_MajorFault.info[0])CLR(Logix_Status.Val_MajorFault.info[1])CLR(Logix_Status.Val_MajorFault.info[2])CLR(Logix_Status.Val_MajorFault.info[3])CLR(Logix_Status.Val_MajorFault.info[4])CLR(Logix_Status.Val_MajorFault.info[5])CLR(Logix_Status.Val_MajorFault.info[6])CLR(Logix_Status.Val_MajorFault.info[7]);
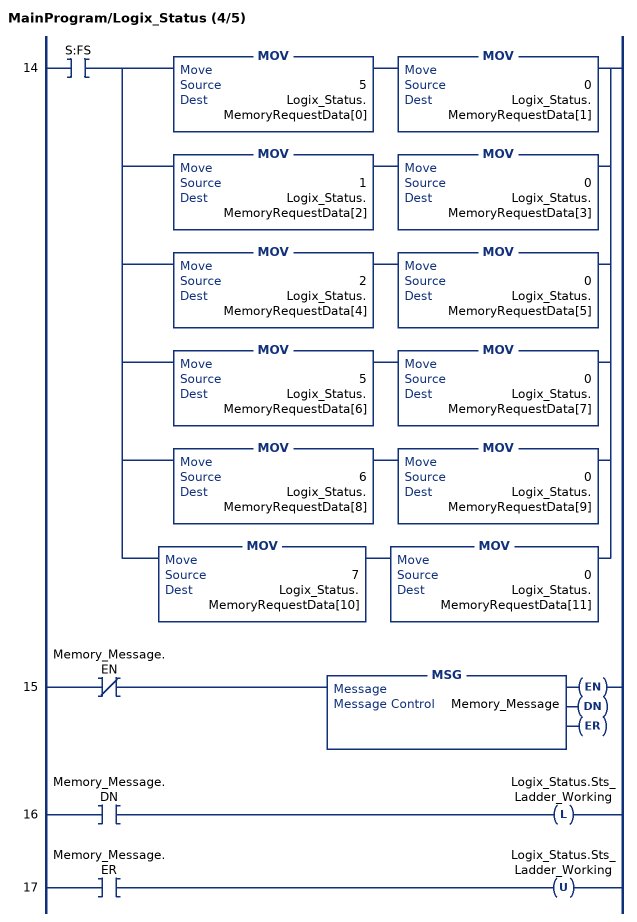
   14: XIC(S:FS)[MOV(5,Logix_Status.MemoryRequestData[0]) MOV(0,Logix_Status.MemoryRequestData[1]) ,MOV(1,Logix_Status.MemoryRequestData[2]) MOV(0,Logix_Status.MemoryRequestData[3]) ,MOV(2,Logix_Status.MemoryRequestData[4]) MOV(0,Logix_Status.MemoryRequestData[5]) ,MOV(5,Logix_Status.MemoryRequestData[6]) MOV(0,Logix_Status.MemoryRequestData[7]) ,MOV(6,Logix_Status.MemoryRequestData[8]) MOV(0,Logix_Status.MemoryRequestData[9]) ,MOV(7,Logix_Status.MemoryRequestData[10]) MOV(0,Logix_Status.MemoryRequestData[11]) ];
   15: XIO(Memory_Message.EN)MSG(Memory_Message);
   16: XIC(Memory_Message.DN)OTL(Logix_Status.Sts_Ladder_Working);
   17: XIC(Memory_Message.ER)OTU(Logix_Status.Sts_Ladder_Working);
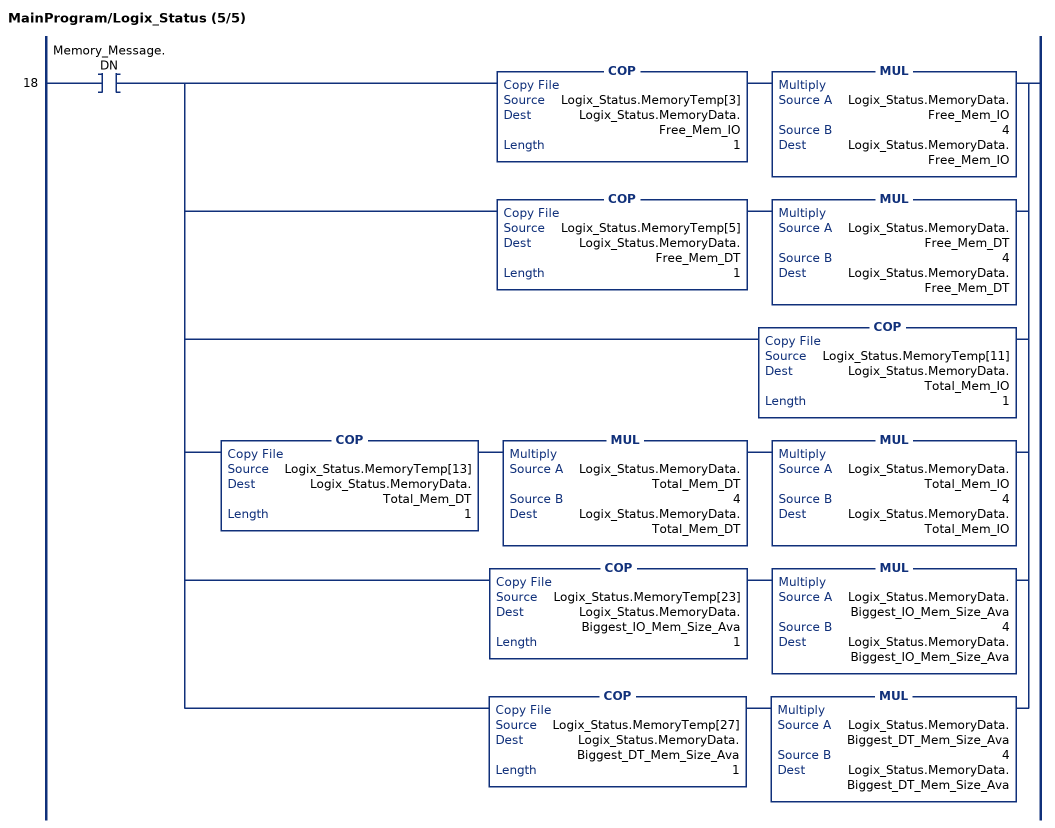
   18: XIC(Memory_Message.DN)[COP(Logix_Status.MemoryTemp[3],Logix_Status.MemoryData.Free_Mem_IO,1) MUL(Logix_Status.MemoryData.Free_Mem_IO,4,Logix_Status.MemoryData.Free_Mem_IO) ,COP(Logix_Status.MemoryTemp[5],Logix_Status.MemoryData.Free_Mem_DT,1) MUL(Logix_Status.MemoryData.Free_Mem_DT,4,Logix_Status.MemoryData.Free_Mem_DT) ,COP(Logix_Status.MemoryTemp[11],Logix_Status.MemoryData.Total_Mem_IO,1) ,COP(Logix_Status.MemoryTemp[13],Logix_Status.MemoryData.Total_Mem_DT,1) MUL(Logix_Status.MemoryData.Total_Mem_DT,4,Logix_Status.MemoryData.Total_Mem_DT) MUL(Logix_Status.MemoryData.Total_Mem_IO,4,Logix_Status.MemoryData.Total_Mem_IO) ,COP(Logix_Status.MemoryTemp[23],Logix_Status.MemoryData.Biggest_IO_Mem_Size_Ava,1) MUL(Logix_Status.MemoryData.Biggest_IO_Mem_Size_Ava,4,Logix_Status.MemoryData.Biggest_IO_Mem_Size_Ava) ,COP(Logix_Status.MemoryTemp[27],Logix_Status.MemoryData.Biggest_DT_Mem_Size_Ava,1) MUL(Logix_Status.MemoryData.Biggest_DT_Mem_Size_Ava,4,Logix_Status.MemoryData.Biggest_DT_Mem_Size_Ava) ];
END_ROUTINE

ROUTINE Main_Seq   (* structured text *)
   (*SECOND PULSE*)
   TON.PRE	:=1000;
   TON.TimerEnable	:=1;
   TONR(TON );
   R_TRIG.InputBit :=TON.DN ;
   OSRI( R_TRIG);
   _SEC_P  := R_TRIG.OutputBit;
   TON.Reset := _SEC_P;
   
   IF  _SEC_P      THEN
   	SEC_TEST:=SEC_TEST+1;
       _SEC_P_2 := 1;         (* we made it *)
   END_IF;
   
   
   
   (*MINUTES PULSE*)
   TON_MIN.PRE	:=60000;
   TON_MIN.TimerEnable	:=1;
   TONR(TON_MIN );
   RTRIG_MIN.InputBit :=TON_MIN.DN ;
   OSRI( RTRIG_MIN);
   _MIN_P  := RTRIG_MIN.OutputBit;
   TON_MIN.Reset := _MIN_P;
   
   IF  _MIN_P      THEN
   	MIN_TEST:=MIN_TEST+1;
   
   END_IF;
   
   (*
   IF HMI_PLANT.STOP THEN
   	HMI_P3_SHUTDOWN:=1;
   END_IF;
   *)
   
   IF HMI_PLANT.STOP OR PLANT_CRITICAL_SD.ON THEN
   	HMI_P3_SHUTDOWN:=1;
   END_IF;
   
   
   (*TMP HIGH*)
   IF HMI_DPIT301.Hty THEN
   	HMI_TMP_HIGH:= HMI_DPIT301.AH;
   ELSE
   	HMI_TMP_HIGH:= HMI_DPSH301.Alarm;
   END_IF;
   
   P6_P602_AUTOINP.ON := _P602_AutoInp;
   
   _ON_ENTRY := _LAST_STATE <> HMI_P3_STATE;
   
   R_TRIG_BW.InputBit :=HMI_P3_STATE =13;
   OSRI( R_TRIG_BW);
   (*
   IF R_TRIG_BW.OutputBit THEN
   	HMI_BW_CNT:= HMI_BW_CNT+1;
   END_IF;
   *)
   (*
   IF HMI_LIT401.AH AND HMI_P3_SHUTDOWN  THEN
   	HMI_P3_STATE:=1;
   END_IF;
   *)
   
   (*
   if S:FS then
   	HMI_P3_STATE := 1;
   end_if;
   *)
   
   
   IF HMI_LIT401.AH AND HMI_P3_STATE > 1 THEN
   	HMI_P3_STATE:=99;
   END_IF;
   
   
   (*-----------WRITE FAULT CONDITION--------------*)
   
   CASE HMI_P3_STATE OF
   	1:(*PLANT IN STANDBY*)
   		_LAST_STATE:= HMI_P3_STATE;
   
   		_MV301_AutoInp			:=0;
   		_MV302_AutoInp			:=0;
   		_MV303_AutoInp			:=0;
   		_MV304_AutoInp			:=0;
   		_P_UF_FEED_DUTY_AutoInp	:=0;
   		_P602_AutoInp			:=0;
   		_P_NAOCL_UF_DUTY_AutoInp:=0;
   
   		HMI_UF_REFILL_SEC		:=0;
   		HMI_UF_FILTRATION_MIN	:=0;
   		HMI_BACKWASH_SEC		:=0;
   		HMI_CIP_CLEANING_SEC	:=0;
   		HMI_DRAIN_SEC			:=0;
   		HMI_P3_SHUTDOWN			:=0;
   
   		IF HMI_P3_PERMISSIVE.ON AND HMI_PLANT.START THEN
   			HMI_P3_STATE:=2;
   		END_IF;
   
   	2:(*MV304, OPEN UF DRAIN VALVE*)
   		_LAST_STATE:= HMI_P3_STATE;
   
   		_MV301_AutoInp			:=0;
   		_MV302_AutoInp			:=0;
   		_MV303_AutoInp			:=0;
   		_MV304_AutoInp			:=NOT HMI_LIT301.ALL AND NOT HMI_LIT401.AH  ;
   		_P_UF_FEED_DUTY_AutoInp	:=0;
   		_P602_AutoInp			:=0;
   		_P_NAOCL_UF_DUTY_AutoInp:=0;
   
   		HMI_UF_REFILL_SEC		:=0;
   		HMI_UF_FILTRATION_MIN	:=0;
   		HMI_BACKWASH_SEC		:=0;
   		HMI_CIP_CLEANING_SEC	:=0;
   		HMI_DRAIN_SEC			:=0;
   
   		IF  HMI_MV304.Status=2 OR _NEXT THEN
   			_NEXT :=0;
   			HMI_P3_STATE:=3;
   		END_IF;
   
   	3:(*P30X , START UF FEED PUMP*)
   		_LAST_STATE:= HMI_P3_STATE;
   
   		_MV301_AutoInp			:=0;
   		_MV302_AutoInp			:=0;
   		_MV303_AutoInp			:=0;
   		_MV304_AutoInp			:=1;
   		_P_UF_FEED_DUTY_AutoInp	:=1;
   		_P602_AutoInp			:=0;
   		_P_NAOCL_UF_DUTY_AutoInp:=0;
   
   		HMI_UF_REFILL_SEC		:=0;
   		HMI_UF_FILTRATION_MIN	:=0;
   		HMI_BACKWASH_SEC		:=0;
   		HMI_CIP_CLEANING_SEC	:=0;
   		HMI_DRAIN_SEC			:=0;
   
   		IF  HMI_P_UF_FEED_DUTY.Pump_Running OR _NEXT THEN
   			_NEXT :=0;
   			HMI_P3_STATE:=4;
   		END_IF;
   
   	4:(*REFILLING FOR PRESET TIMER*)
   		_LAST_STATE:= HMI_P3_STATE;
   
   		_MV301_AutoInp			:=0;
   		_MV302_AutoInp			:=0;
   		_MV303_AutoInp			:=0;
   		_MV304_AutoInp			:=1;
   		_P_UF_FEED_DUTY_AutoInp	:=1;
   		_P602_AutoInp			:=0;
   		_P_NAOCL_UF_DUTY_AutoInp:=0;
   
   		HMI_UF_FILTRATION_MIN	:=0;
   		HMI_BACKWASH_SEC		:=0;
   		HMI_CIP_CLEANING_SEC	:=0;
   		HMI_DRAIN_SEC			:=0;
   
   		IF _SEC_P THEN
   			HMI_UF_REFILL_SEC:=HMI_UF_REFILL_SEC+1;
   			IF HMI_UF_REFILL_SEC>HMI_UF_REFILL_SEC_SP OR _NEXT THEN
   				_NEXT :=0;
   				HMI_P3_STATE:=5;
   			END_IF;
   		END_IF;
   
   	5:(*MV302, OPEN RO FEED VALVE VALVE*)
   		_LAST_STATE:= HMI_P3_STATE;
   
   		_MV301_AutoInp			:=0;
   		_MV302_AutoInp			:=1;
   		_MV303_AutoInp			:=0;
   		_MV304_AutoInp			:=1;
   		_P_UF_FEED_DUTY_AutoInp	:=1;
   		_P602_AutoInp			:=0;
   		_P_NAOCL_UF_DUTY_AutoInp:=0;
   
   		HMI_UF_REFILL_SEC		:=0;
   		HMI_UF_FILTRATION_MIN	:=0;
   		HMI_BACKWASH_SEC		:=0;
   		HMI_CIP_CLEANING_SEC	:=0;
   		HMI_DRAIN_SEC			:=0;
   
   		IF HMI_MV302.Status =2 OR _NEXT THEN
   			_NEXT :=0;
   			HMI_P3_STATE:=6;
   		END_IF;
   
   	6:(*MV304, CLOSE UF DRAIN VALVE*)
   		_LAST_STATE:= HMI_P3_STATE;
   
   		_MV301_AutoInp			:=0;
   		_MV302_AutoInp			:=1;
   		_MV303_AutoInp			:=0;
   		_MV304_AutoInp			:=0;
   		_P_UF_FEED_DUTY_AutoInp	:=1;
   		_P602_AutoInp			:=0;
   		_P_NAOCL_UF_DUTY_AutoInp:=0;
   
   		HMI_UF_REFILL_SEC		:=0;
   		HMI_UF_FILTRATION_MIN	:=0;
   		HMI_BACKWASH_SEC		:=0;
   		HMI_CIP_CLEANING_SEC	:=0;
   		HMI_DRAIN_SEC			:=0;
   
   		IF HMI_MV304.Status =1 OR _NEXT THEN
   			_NEXT :=0;
   			HMI_P3_STATE:=7;
   		END_IF;
   
   	7:(*FILTRATION FOR PRESET TIMER*)
   		_LAST_STATE:= HMI_P3_STATE;
   
   		_MV301_AutoInp			:=0;
   		_MV302_AutoInp			:=1;
   		_MV303_AutoInp			:=0;
   		_MV304_AutoInp			:=0;
   		_P_UF_FEED_DUTY_AutoInp	:=1;
   		_P602_AutoInp			:=0;
   		_P_NAOCL_UF_DUTY_AutoInp:=0;
   
   		HMI_UF_REFILL_SEC		:=0;
   
   		HMI_BACKWASH_SEC		:=0;
   		HMI_CIP_CLEANING_SEC	:=0;
   		HMI_DRAIN_SEC			:=0;
   
   		IF HMI_TMP_HIGH THEN
   			HMI_P3_STATE:=8;
   		ELSE
   			IF _MIN_P THEN
   				HMI_UF_FILTRATION_MIN:= HMI_UF_FILTRATION_MIN+1;
   
   			END_IF;
   		END_IF;
   
   		IF HMI_UF_FILTRATION_MIN>=HMI_UF_FILTRATION_MIN_SP OR _NEXT THEN
   			_NEXT :=0;
   			HMI_P3_STATE:=8;
   		END_IF;
   
   
   		IF  HMI_P3_SHUTDOWN AND HMI_LIT401.AH THEN
   			_NEXT :=0;
   			HMI_P3_STATE:=8;
   
   		END_IF;
   
   
   	8:(*STOP UF FEED PUMP*)
   		_LAST_STATE:= HMI_P3_STATE;
   
   		_MV301_AutoInp			:=0;
   		_MV302_AutoInp			:=1;
   		_MV303_AutoInp			:=0;
   		_MV304_AutoInp			:=0;
   		_P_UF_FEED_DUTY_AutoInp	:=0;
   		_P602_AutoInp			:=0;
   		_P_NAOCL_UF_DUTY_AutoInp:=0;
   
   		HMI_UF_REFILL_SEC		:=0;
   		HMI_UF_FILTRATION_MIN	:=0;
   		HMI_BACKWASH_SEC		:=0;
   		HMI_CIP_CLEANING_SEC	:=0;
   		HMI_DRAIN_SEC			:=0;
   
   		IF NOT HMI_P_UF_FEED_DUTY.Pump_Running OR _NEXT THEN
   			_NEXT :=0;
   			HMI_P3_STATE:=9;
   		END_IF;
   
   	9:(*MV302, CLOSE RO FEED VALVE*)
   		_LAST_STATE:= HMI_P3_STATE;
   
   		_MV301_AutoInp			:=0;
   		_MV302_AutoInp			:=0;
   		_MV303_AutoInp			:=0;
   		_MV304_AutoInp			:=0;
   		_P_UF_FEED_DUTY_AutoInp	:=0;
   		_P602_AutoInp			:=0;
   		_P_NAOCL_UF_DUTY_AutoInp:=0;
   
   		HMI_UF_REFILL_SEC		:=0;
   		HMI_UF_FILTRATION_MIN	:=0;
   		HMI_BACKWASH_SEC		:=0;
   		HMI_CIP_CLEANING_SEC	:=0;
   		HMI_DRAIN_SEC			:=0;
   
   		IF HMI_P3_SHUTDOWN THEN
   			HMI_P3_STATE:=1;
   
   		ELSIF HMI_MV302.Status=1 OR _NEXT AND (NOT HMI_P3_SHUTDOWN) THEN
   			_NEXT :=0;
   			HMI_P3_STATE:=10;
   
   		END_IF;
   
   	10:(*MV301 MV303, OPEN BW VALVE, DRAIN VALVE*)
   		_LAST_STATE:= HMI_P3_STATE;
   
   		_MV301_AutoInp			:=1;
   		_MV302_AutoInp			:=0;
   		_MV303_AutoInp			:=1;
   		_MV304_AutoInp			:=0;
   		_P_UF_FEED_DUTY_AutoInp	:=0;
   		_P602_AutoInp			:=0;
   		_P_NAOCL_UF_DUTY_AutoInp:=0;
   
   		HMI_UF_REFILL_SEC		:=0;
   		HMI_UF_FILTRATION_MIN	:=0;
   		HMI_BACKWASH_SEC		:=0;
   		HMI_CIP_CLEANING_SEC	:=0;
   		HMI_DRAIN_SEC			:=0;
   
   		IF HMI_MV301.Status=2 AND HMI_MV303.Status=2 OR _NEXT THEN
   			_NEXT :=0;
   			HMI_P3_STATE:=11;
   		END_IF;
   
   	11:(*P602, START BW PUMP*)
   		_LAST_STATE:= HMI_P3_STATE;
   
   		_MV301_AutoInp			:=1;
   		_MV302_AutoInp			:=0;
   		_MV303_AutoInp			:=1;
   		_MV304_AutoInp			:=0;
   		_P_UF_FEED_DUTY_AutoInp	:=0;
   		_P602_AutoInp			:=1;
   		_P_NAOCL_UF_DUTY_AutoInp:=0;
   
   		HMI_UF_REFILL_SEC		:=0;
   		HMI_UF_FILTRATION_MIN	:=0;
   		HMI_BACKWASH_SEC		:=0;
   		HMI_CIP_CLEANING_SEC	:=0;
   		HMI_DRAIN_SEC			:=0;
   
   		IF HMI_P602.Status=2 OR _NEXT THEN
   			_NEXT :=0;
   			HMI_P3_STATE:=12;
   		END_IF;
   
   	12:(*BACKWASH*)
   		_LAST_STATE:= HMI_P3_STATE;
   
   		_MV301_AutoInp			:=1;
   		_MV302_AutoInp			:=0;
   		_MV303_AutoInp			:=1;
   		_MV304_AutoInp			:=0;
   		_P_UF_FEED_DUTY_AutoInp	:=0;
   		_P602_AutoInp			:=1;
   		_P_NAOCL_UF_DUTY_AutoInp:=0;
   
   		HMI_UF_REFILL_SEC		:=0;
   		HMI_UF_FILTRATION_MIN	:=0;
   
   		HMI_CIP_CLEANING_SEC	:=0;
   		HMI_DRAIN_SEC			:=0;
   
   		IF _SEC_P THEN
   			HMI_BACKWASH_SEC:= HMI_BACKWASH_SEC+1;
   			IF HMI_BACKWASH_SEC> HMI_BACKWASH_SEC_SP OR _NEXT THEN
   				_NEXT :=0;
   					HMI_BW_CNT:= HMI_BW_CNT+1;
   				HMI_P3_STATE:=13;
   			END_IF;
   		END_IF;
   
   	13: (*P602, STOP BW PUMP*)
   	(*F _ON_ENTRY THEN
   			HMI_BW_CNT:= HMI_BW_CNT+1;
   		END_IF;
   		*)
   
   		_LAST_STATE:= HMI_P3_STATE;
   
   
   
   		_MV301_AutoInp			:=1;
   		_MV302_AutoInp			:=0;
   		_MV303_AutoInp			:=1;
   		_MV304_AutoInp			:=0;
   		_P_UF_FEED_DUTY_AutoInp	:=0;
   		_P602_AutoInp			:=0;
   		_P_NAOCL_UF_DUTY_AutoInp:=0;
   
   		HMI_UF_REFILL_SEC		:=0;
   		HMI_UF_FILTRATION_MIN	:=0;
   		HMI_BACKWASH_SEC		:=0;
   		HMI_CIP_CLEANING_SEC	:=0;
   		HMI_DRAIN_SEC			:=0;
   
   		IF HMI_P602.Status=1 OR _NEXT THEN
   			(*HMI_BW_CNT:= HMI_BW_CNT+1;*)
   		(*	IF _NEXT THEN*)
   
   				HMI_P3_STATE:=14; (* CIP CLEANING AFTER 6 TIMES BW*)
   		(*	ELSIF _NEXT THEN
   				_NEXT :=0;
   				HMI_P3_STATE:=14;
   			END_IF;	*)
   		END_IF;
   
   	14: (*MV301 CLOSE BW *)
   		_LAST_STATE:= HMI_P3_STATE;
   
   		_MV301_AutoInp			:=0;
   		_MV302_AutoInp			:=0;
   		_MV303_AutoInp			:=1;
   		_MV304_AutoInp			:=0;
   		_P_UF_FEED_DUTY_AutoInp	:=0;
   		_P602_AutoInp			:=0;
   		_P_NAOCL_UF_DUTY_AutoInp:=0;
   
   		HMI_UF_REFILL_SEC		:=0;
   		HMI_UF_FILTRATION_MIN	:=0;
   		HMI_BACKWASH_SEC		:=0;
   		HMI_CIP_CLEANING_SEC	:=0;
   		HMI_DRAIN_SEC			:=0;
   
   		IF HMI_MV301.Status=1 OR _NEXT THEN
   			_NEXT:=0;
   			HMI_P3_STATE:=15;
   		END_IF;
   
   	15: (*MV304,OPEN UF DRAIN VALVE*)
   		_LAST_STATE:= HMI_P3_STATE;
   
   		_MV301_AutoInp			:=0;
   		_MV302_AutoInp			:=0;
   		_MV303_AutoInp			:=1;
   		_MV304_AutoInp			:=1;
   		_P_UF_FEED_DUTY_AutoInp	:=0;
   		_P602_AutoInp			:=0;
   		_P_NAOCL_UF_DUTY_AutoInp:=0;
   
   		HMI_UF_REFILL_SEC		:=0;
   		HMI_UF_FILTRATION_MIN	:=0;
   		HMI_BACKWASH_SEC		:=0;
   		HMI_CIP_CLEANING_SEC	:=0;
   		HMI_DRAIN_SEC			:=0;
   
   		IF HMI_MV304.Status=2 OR _NEXT THEN
   			_NEXT:=0;
   			HMI_P3_STATE:=16;
   		END_IF;
   
   	16: (*DRAINING*)
   		_LAST_STATE:= HMI_P3_STATE;
   
   		_MV301_AutoInp			:=0;
   		_MV302_AutoInp			:=0;
   		_MV303_AutoInp			:=1;
   		_MV304_AutoInp			:=1;
   		_P_UF_FEED_DUTY_AutoInp	:=0;
   		_P602_AutoInp			:=0;
   		_P_NAOCL_UF_DUTY_AutoInp:=0;
   
   		HMI_UF_REFILL_SEC		:=0;
   		HMI_UF_FILTRATION_MIN	:=0;
   		HMI_BACKWASH_SEC		:=0;
   		HMI_CIP_CLEANING_SEC	:=0;
   
   		IF _SEC_P THEN
   			HMI_DRAIN_SEC:=HMI_DRAIN_SEC+1;
   			IF HMI_DRAIN_SEC>HMI_DRAIN_SEC_SP OR _NEXT THEN
   				_NEXT:=0;
   				HMI_P3_STATE:=4;
   			END_IF;
   		END_IF;
   
   (*-------------------CIP--------------------- *)
   	17: (*P20X, START NAOCL DOSING PUMP*)
   		_MV301_AutoInp			:=1;
   		_MV302_AutoInp			:=0;
   		_MV303_AutoInp			:=1;
   		_MV304_AutoInp			:=0;
   		_P_UF_FEED_DUTY_AutoInp	:=0;
   		_P602_AutoInp			:=0;
   		_P_NAOCL_UF_DUTY_AutoInp:=1;
   
   		HMI_UF_REFILL_SEC		:=0;
   		HMI_UF_FILTRATION_MIN	:=0;
   		HMI_BACKWASH_SEC		:=0;
   		HMI_CIP_CLEANING_SEC	:=0;
   		HMI_DRAIN_SEC			:=0;
   
   		IF HMI_P_NAOCL_UF_DUTY.Pump_Running OR _NEXT THEN
   			_NEXT:=0;
   			HMI_P3_STATE:=18;
   		END_IF;
   
   	18: (*CIP CLEANING*)
   		_MV301_AutoInp			:=1;
   		_MV302_AutoInp			:=0;
   		_MV303_AutoInp			:=1;
   		_MV304_AutoInp			:=0;
   		_P_UF_FEED_DUTY_AutoInp	:=0;
   		_P602_AutoInp			:=0;
   		_P_NAOCL_UF_DUTY_AutoInp:=1;
   
   		HMI_UF_REFILL_SEC		:=0;
   		HMI_UF_FILTRATION_MIN	:=0;
   		HMI_BACKWASH_SEC		:=0;
   
   		HMI_DRAIN_SEC			:=0;
   
   		IF _SEC_P THEN
   			HMI_CIP_CLEANING_SEC:=HMI_CIP_CLEANING_SEC+1;
   			IF HMI_CIP_CLEANING_SEC>HMI_CIP_CLEANING_SEC_SP OR _NEXT THEN
   				_NEXT:=0;
   				HMI_P3_STATE:=19;
   			END_IF;
   		END_IF;
   
   	19: (*P207/8 , STOP NAOCL DOSING PUMP*)
   		_MV301_AutoInp			:=1;
   		_MV302_AutoInp			:=0;
   		_MV303_AutoInp			:=1;
   		_MV304_AutoInp			:=0;
   		_P_UF_FEED_DUTY_AutoInp	:=0;
   		_P602_AutoInp			:=0;
   		_P_NAOCL_UF_DUTY_AutoInp:=0;
   
   		HMI_UF_REFILL_SEC		:=0;
   		HMI_UF_FILTRATION_MIN	:=0;
   		HMI_BACKWASH_SEC		:=0;
   
   		HMI_DRAIN_SEC			:=0;
   
   		IF NOT HMI_P_NAOCL_UF_DUTY.Pump_Running OR _NEXT THEN
   				_NEXT:=0;
   				HMI_P3_STATE:=14;
   		END_IF;
   
   	99: (*STANDBY*)
   		_MV301_AutoInp			:=00;
   		_MV302_AutoInp			:=0;
   		_MV303_AutoInp			:=0;
   		_MV304_AutoInp			:=0;
   		_P_UF_FEED_DUTY_AutoInp	:=0;
   		_P602_AutoInp			:=0;
   		_P_NAOCL_UF_DUTY_AutoInp:=0;
   
   		HMI_UF_REFILL_SEC		:=0;
   		HMI_UF_FILTRATION_MIN	:=0;
   		HMI_BACKWASH_SEC		:=0;
   		HMI_CIP_CLEANING_SEC	:=0;
   		HMI_DRAIN_SEC			:=0;
   
   		IF  (HMI_LIT401.AL AND NOT HMI_P3_SHUTDOWN ) OR HMI_PLANT.START THEN
   			HMI_P3_STATE:=2;
   		ELSIF HMI_LIT401.AH AND HMI_P3_SHUTDOWN THEN
   			HMI_P3_STATE:=1;
   		END_IF;
   
   
   
   ELSE
   	HMI_P3_STATE:=1;
   END_CASE;
   
   
   
   
   
   
END_ROUTINE

ROUTINE MainRoutine   (* ladder *)
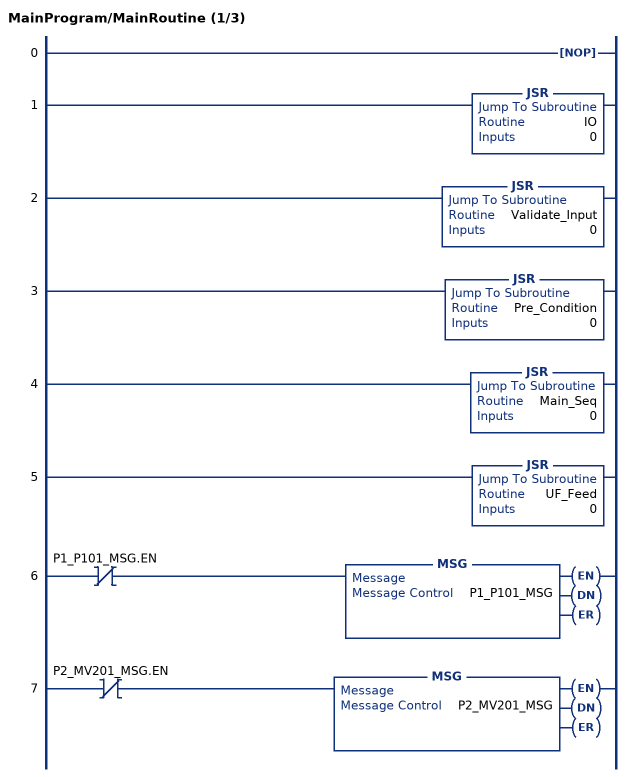
   0: NOP();
   1: JSR(IO,0);
   2: JSR(Validate_Input,0);
   3: JSR(Pre_Condition,0);
   4: JSR(Main_Seq,0);
   5: JSR(UF_Feed,0);
   6: XIO(P1_P101_MSG.EN)MSG(P1_P101_MSG);
   7: XIO(P2_MV201_MSG.EN)MSG(P2_MV201_MSG);
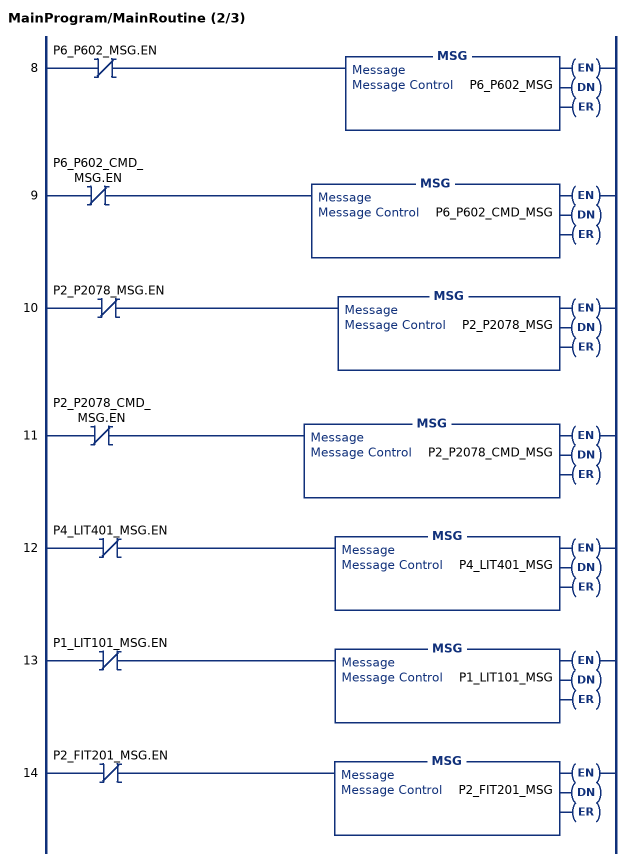
   8: XIO(P6_P602_MSG.EN)MSG(P6_P602_MSG);
   9: XIO(P6_P602_CMD_MSG.EN)MSG(P6_P602_CMD_MSG);
   10: XIO(P2_P2078_MSG.EN)MSG(P2_P2078_MSG);
   11: XIO(P2_P2078_CMD_MSG.EN)MSG(P2_P2078_CMD_MSG);
   12: XIO(P4_LIT401_MSG.EN)MSG(P4_LIT401_MSG);
   13: XIO(P1_LIT101_MSG.EN)MSG(P1_LIT101_MSG);
   14: XIO(P2_FIT201_MSG.EN)MSG(P2_FIT201_MSG);
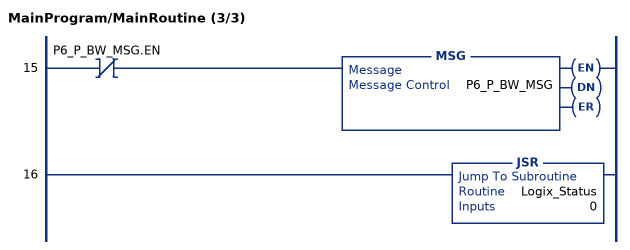
   15: XIO(P6_P_BW_MSG.EN)MSG(P6_P_BW_MSG);
   16: JSR(Logix_Status,0);
END_ROUTINE

ROUTINE Pre_Condition   (* structured text *)
   (*RESET ALL INSTRUMENT*)
   IF HMI_PLANT_RESET.ON THEN
   	HMI_MV301.Reset	:=1;
   	HMI_MV302.Reset	:=1;
   	HMI_MV303.Reset	:=1;
   	HMI_MV304.Reset	:=1;
   	HMI_P301.Reset	:=1;
   	HMI_P302.Reset	:=1;
   END_IF;
   
   (*ALL INSTRUMENT IN AUTO MODE*)
   IF HMI_PLANT_AUTO.ON THEN
   	HMI_MV301.Auto	:=1;
   	HMI_MV302.Auto	:=1;
   	HMI_MV303.Auto	:=1;
   	HMI_MV304.Auto	:=1;
   	HMI_P301.Auto	:=1;
   	HMI_P302.Auto	:=1;
   END_IF;
   
   (*ALL INSTRUMENT IN MANUAL MODE*)
   IF HMI_PLANT_AUTO.OFF THEN
   	HMI_MV301.Auto	:=0;
   	HMI_MV302.Auto	:=0;
   	HMI_MV303.Auto	:=0;
   	HMI_MV304.Auto	:=0;
   	HMI_P301.Auto	:=0;
   	HMI_P302.Auto	:=0;
   END_IF;
   
   (*P3 PERMISSIVE*)
   HMI_P3_PERMISSIVE.ON 	:=  HMI_MV301.Avl AND HMI_MV302.Avl AND HMI_MV303.Avl AND HMI_MV304.Avl AND (HMI_P301.Avl OR HMI_P302.Avl);
   
   
   (*Enable Flow Totalising*)
   _FIT301_Tot_Enb	:= HMI_P301.status=2 OR HMI_P302.status=2;
   
   TON_FIT301_P1_TM.PRE 			:= 	6*1000;
   TON_FIT301_P1_TM.TimerEnable 	:=  HMI_FIT301.ALL AND HMI_P301.STATUS=2 ;
   TONR(TON_FIT301_P1_TM);
   
   TON_FIT301_P2_TM.PRE 			:= 	6*1000;
   TON_FIT301_P2_TM.TimerEnable 	:=  HMI_FIT301.ALL AND HMI_P302.STATUS=2 ;
   TONR(TON_FIT301_P2_TM);
   
   (*P301 Permissive*)
   HMI_P301.Permissive.0 	:= NOT HMI_LIT301.ALL;
   HMI_P301.Permissive.1 	:= NOT HMI_LIT401.AHH;
   HMI_P301.Permissive.2 	:= HMI_MV302.STATUS=2 OR HMI_MV304.STATUS=2;
   HMI_P301.Permissive.3 	:= 1;
   HMI_P301.Permissive.4 	:= 1;
   HMI_P301.Permissive.5 	:= 1;
   HMI_P301.Permissive.6 	:= 1;
   HMI_P301.Permissive.7 	:= 1;
   HMI_P301.Permissive.8 	:= 1;
   HMI_P301.Permissive.9 	:= 1;
   HMI_P301.Permissive.10 	:= 1;
   HMI_P301.Permissive.11 	:= 1;
   HMI_P301.Permissive.12 	:= 1;
   HMI_P301.Permissive.13	:= 1;
   HMI_P301.Permissive.14	:= 1;
   HMI_P301.Permissive.15 	:= 1;
   
   HMI_P301_MSG.PERMISSIVE1 := HMI_P301.Permissive.0;
   HMI_P301_MSG.PERMISSIVE2 := HMI_P301.Permissive.1;
   HMI_P301_MSG.PERMISSIVE3 := HMI_P301.Permissive.2;
   HMI_P301_MSG.PERMISSIVE4 := 0;
   HMI_P301_MSG.PERMISSIVE5 := 0;
   
   (*P302 Permissive*)
   HMI_P302.Permissive.0 	:= NOT HMI_LIT301.ALL;
   HMI_P302.Permissive.1 	:= NOT HMI_LIT401.AHH;
   HMI_P302.Permissive.2 	:= HMI_MV302.STATUS=2 OR HMI_MV304.STATUS=2;
   HMI_P302.Permissive.3 	:= 1;
   HMI_P302.Permissive.4 	:= 1;
   HMI_P302.Permissive.5 	:= 1;
   HMI_P302.Permissive.6 	:= 1;
   HMI_P302.Permissive.7 	:= 1;
   HMI_P302.Permissive.8 	:= 1;
   HMI_P302.Permissive.9 	:= 1;
   HMI_P302.Permissive.10 	:= 1;
   HMI_P302.Permissive.11 	:= 1;
   HMI_P302.Permissive.12 	:= 1;
   HMI_P302.Permissive.13	:= 1;
   HMI_P302.Permissive.14	:= 1;
   HMI_P302.Permissive.15 	:= 1;
   
   HMI_P302_MSG.PERMISSIVE1 := HMI_P302.Permissive.0;
   HMI_P302_MSG.PERMISSIVE2 := HMI_P302.Permissive.1;
   HMI_P302_MSG.PERMISSIVE3 := HMI_P302.Permissive.2;
   HMI_P302_MSG.PERMISSIVE4 := 0;
   HMI_P302_MSG.PERMISSIVE5 := 0;
   
   (*-------------------------------------------------------------------------------------*)
   (*P301 Shutdown*)
   HMI_P301.SD.0 	:= HMI_LIT301.ALL;
   HMI_P301.SD.1 	:= HMI_LIT401.AHH;
   HMI_P301.SD.2 	:= HMI_PSH301.Alarm;
   HMI_P301.SD.3 	:= 0;(*TON_FIT301_P1_TM.DN;*)
   HMI_P301.SD.4 	:= HMI_P301.STATUS =2 AND HMI_MV302.STATUS<>2 AND HMI_MV304.STATUS<>2;
   HMI_P301.SD.5 	:= 0;
   HMI_P301.SD.6 	:= 0;
   HMI_P301.SD.7 	:= 0;
   HMI_P301.SD.8 	:= 0;
   HMI_P301.SD.9 	:= 0;
   HMI_P301.SD.10 	:= 0;
   HMI_P301.SD.11 	:= 0;
   HMI_P301.SD.12 	:= 0;
   HMI_P301.SD.13 	:= 0;
   HMI_P301.SD.14 	:= 0;
   HMI_P301.SD.15 	:= 0;
   
   HMI_P301_MSG.SHUTDOWN1 := HMI_P301.SHUTDOWN.0 ;
   HMI_P301_MSG.SHUTDOWN2 := HMI_P301.SHUTDOWN.1 ;
   HMI_P301_MSG.SHUTDOWN3 := HMI_P301.SHUTDOWN.2 ;
   HMI_P301_MSG.SHUTDOWN4 := HMI_P301.SHUTDOWN.3 ;
   HMI_P301_MSG.SHUTDOWN5 := HMI_P301.SHUTDOWN.4 ;
   
   (*P302 Shutdown*)
   HMI_P302.SD.0 	:= HMI_LIT301.ALL;
   HMI_P302.SD.1 	:= HMI_LIT401.AHH;
   HMI_P302.SD.2 	:= HMI_PSH301.Alarm;
   HMI_P302.SD.3 	:= 0;(*TON_FIT301_P2_TM.DN;*)
   HMI_P302.SD.4 	:= HMI_P302.STATUS =2 AND HMI_MV302.STATUS<>2 AND HMI_MV304.STATUS<>2;
   HMI_P302.SD.5 	:= 0;
   HMI_P302.SD.6 	:= 0;
   HMI_P302.SD.7 	:= 0;
   HMI_P302.SD.8 	:= 0;
   HMI_P302.SD.9 	:= 0;
   HMI_P302.SD.10 	:= 0;
   HMI_P302.SD.11 	:= 0;
   HMI_P302.SD.12 	:= 0;
   HMI_P302.SD.13 	:= 0;
   HMI_P302.SD.14 	:= 0;
   HMI_P302.SD.15 	:= 0;
   
   HMI_P302_MSG.SHUTDOWN1 := HMI_P302.SHUTDOWN.0 ;
   HMI_P302_MSG.SHUTDOWN2 := HMI_P302.SHUTDOWN.1 ;
   HMI_P302_MSG.SHUTDOWN3 := HMI_P302.SHUTDOWN.2 ;
   HMI_P302_MSG.SHUTDOWN4 := HMI_P302.SHUTDOWN.3 ;
   HMI_P302_MSG.SHUTDOWN5 := HMI_P302.SHUTDOWN.4 ;
   
END_ROUTINE

ROUTINE UF_Feed   (* function block diagram *)
   SHEET 1
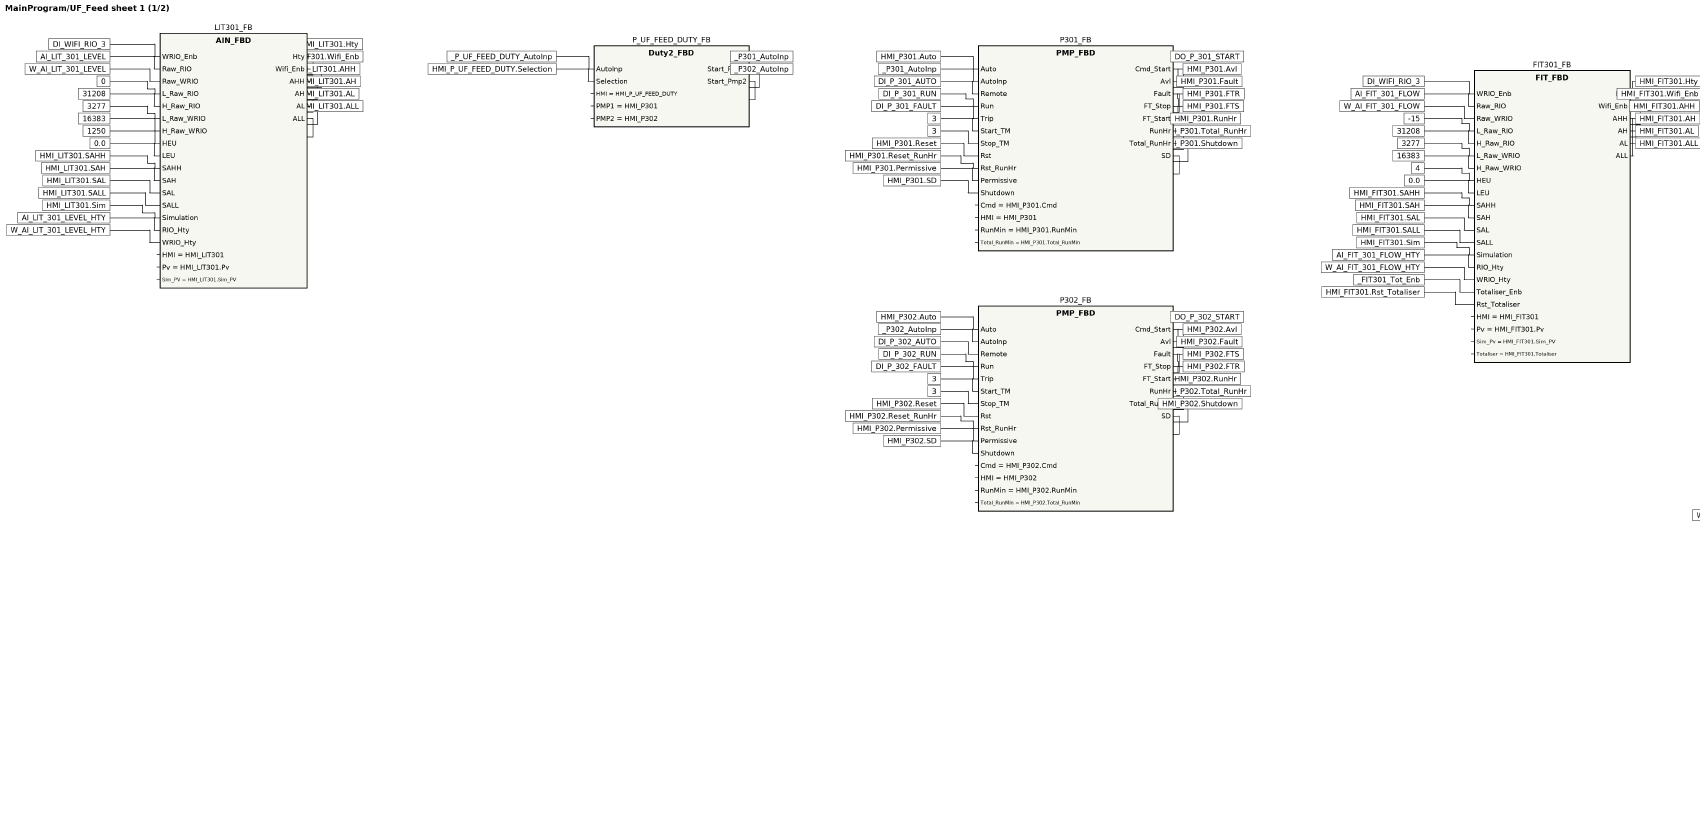
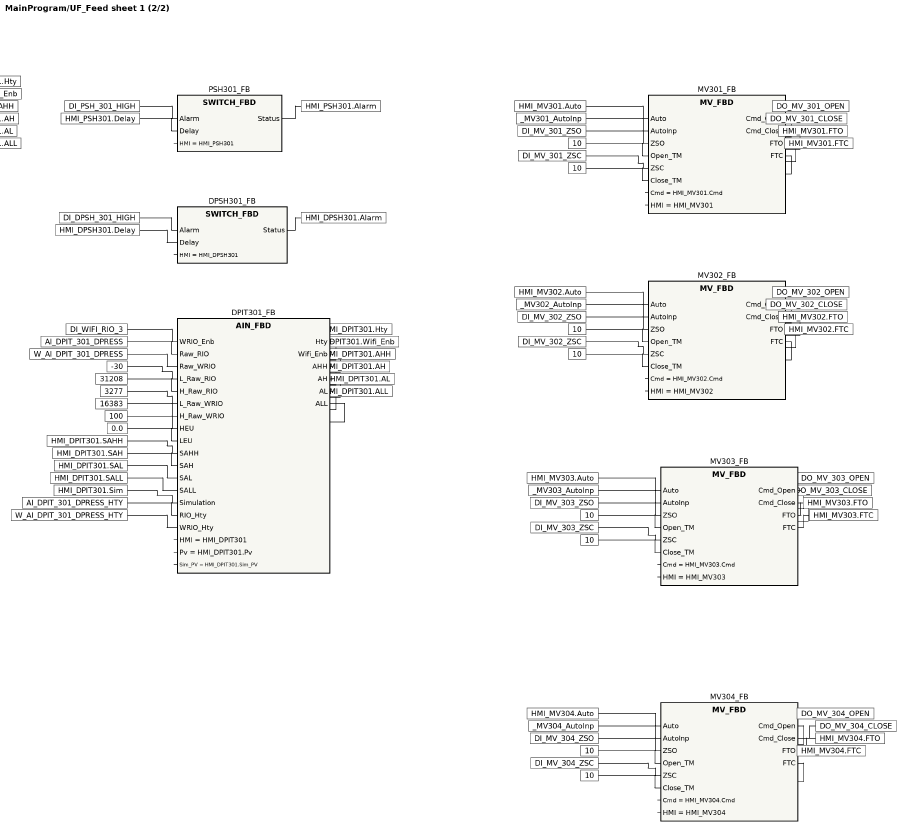
   LIT301_FB : AIN_FBD(WRIO_Enb := DI_WIFI_RIO_3, Raw_RIO := AI_LIT_301_LEVEL, Raw_WRIO := W_AI_LIT_301_LEVEL, L_Raw_RIO := 0, H_Raw_RIO := 31208, L_Raw_WRIO := 3277, H_Raw_WRIO := 16383, HEU := 1250, LEU := 0.0, SAHH := HMI_LIT301.SAHH, SAH := HMI_LIT301.SAH, SAL := HMI_LIT301.SAL, SALL := HMI_LIT301.SALL, Simulation := HMI_LIT301.Sim, RIO_Hty := AI_LIT_301_LEVEL_HTY, WRIO_Hty := W_AI_LIT_301_LEVEL_HTY, HMI := HMI_LIT301, Pv := HMI_LIT301.Pv, Sim_PV := HMI_LIT301.Sim_PV);
   HMI_LIT301.Wifi_Enb := LIT301_FB.Wifi_Enb;
   HMI_LIT301.AHH := LIT301_FB.AHH;
   HMI_LIT301.Hty := LIT301_FB.Hty;
   HMI_LIT301.AH := LIT301_FB.AH;
   HMI_LIT301.AL := LIT301_FB.AL;
   HMI_LIT301.ALL := LIT301_FB.ALL;
   P_UF_FEED_DUTY_FB : Duty2_FBD(AutoInp := _P_UF_FEED_DUTY_AutoInp, Selection := HMI_P_UF_FEED_DUTY.Selection, HMI := HMI_P_UF_FEED_DUTY, PMP1 := HMI_P301, PMP2 := HMI_P302);
   _P301_AutoInp := P_UF_FEED_DUTY_FB.Start_Pmp1;
   _P302_AutoInp := P_UF_FEED_DUTY_FB.Start_Pmp2;
   P301_FB : PMP_FBD(Auto := HMI_P301.Auto, AutoInp := _P301_AutoInp, Remote := DI_P_301_AUTO, Run := DI_P_301_RUN, Trip := DI_P_301_FAULT, Start_TM := 3, Stop_TM := 3, Rst := HMI_P301.Reset, Rst_RunHr := HMI_P301.Reset_RunHr, Permissive := HMI_P301.Permissive, Shutdown := HMI_P301.SD, Cmd := HMI_P301.Cmd, HMI := HMI_P301, RunMin := HMI_P301.RunMin, Total_RunMin := HMI_P301.Total_RunMin);
   P302_FB : PMP_FBD(Auto := HMI_P302.Auto, AutoInp := _P302_AutoInp, Remote := DI_P_302_AUTO, Run := DI_P_302_RUN, Trip := DI_P_302_FAULT, Start_TM := 3, Stop_TM := 3, Rst := HMI_P302.Reset, Rst_RunHr := HMI_P302.Reset_RunHr, Permissive := HMI_P302.Permissive, Shutdown := HMI_P302.SD, Cmd := HMI_P302.Cmd, HMI := HMI_P302, RunMin := HMI_P302.RunMin, Total_RunMin := HMI_P302.Total_RunMin);
   HMI_P301.Total_RunHr := P301_FB.Total_RunHr;
   HMI_P301.Shutdown := P301_FB.SD;
   HMI_P302.Total_RunHr := P302_FB.Total_RunHr;
   HMI_P302.Shutdown := P302_FB.SD;
   DO_P_301_START := P301_FB.Cmd_Start;
   HMI_P301.RunHr := P301_FB.RunHr;
   DO_P_302_START := P302_FB.Cmd_Start;
   HMI_P302.RunHr := P302_FB.RunHr;
   HMI_P301.Fault := P301_FB.Fault;
   HMI_P302.Fault := P302_FB.Fault;
   HMI_P301.Avl := P301_FB.Avl;
   HMI_P301.FTR := P301_FB.FT_Stop;
   HMI_P301.FTS := P301_FB.FT_Start;
   HMI_P302.Avl := P302_FB.Avl;
   HMI_P302.FTS := P302_FB.FT_Stop;
   HMI_P302.FTR := P302_FB.FT_Start;
   FIT301_FB : FIT_FBD(WRIO_Enb := DI_WIFI_RIO_3, Raw_RIO := AI_FIT_301_FLOW, Raw_WRIO := W_AI_FIT_301_FLOW, L_Raw_RIO := -15, H_Raw_RIO := 31208, L_Raw_WRIO := 3277, H_Raw_WRIO := 16383, HEU := 4, LEU := 0.0, SAHH := HMI_FIT301.SAHH, SAH := HMI_FIT301.SAH, SAL := HMI_FIT301.SAL, SALL := HMI_FIT301.SALL, Simulation := HMI_FIT301.Sim, RIO_Hty := AI_FIT_301_FLOW_HTY, WRIO_Hty := W_AI_FIT_301_FLOW_HTY, Totaliser_Enb := _FIT301_Tot_Enb, Rst_Totaliser := HMI_FIT301.Rst_Totaliser, HMI := HMI_FIT301, Pv := HMI_FIT301.Pv, Sim_Pv := HMI_FIT301.Sim_PV, Totaliser := HMI_FIT301.Totaliser);
   HMI_FIT301.Wifi_Enb := FIT301_FB.Wifi_Enb;
   HMI_FIT301.AHH := FIT301_FB.AHH;
   HMI_FIT301.Hty := FIT301_FB.Hty;
   HMI_FIT301.AH := FIT301_FB.AH;
   HMI_FIT301.AL := FIT301_FB.AL;
   HMI_FIT301.ALL := FIT301_FB.ALL;
   PSH301_FB : SWITCH_FBD(Alarm := DI_PSH_301_HIGH, Delay := HMI_PSH301.Delay, HMI := HMI_PSH301);
   DPSH301_FB : SWITCH_FBD(Alarm := DI_DPSH_301_HIGH, Delay := HMI_DPSH301.Delay, HMI := HMI_DPSH301);
   DPIT301_FB : AIN_FBD(WRIO_Enb := DI_WIFI_RIO_3, Raw_RIO := AI_DPIT_301_DPRESS, Raw_WRIO := W_AI_DPIT_301_DPRESS, L_Raw_RIO := -30, H_Raw_RIO := 31208, L_Raw_WRIO := 3277, H_Raw_WRIO := 16383, HEU := 100, LEU := 0.0, SAHH := HMI_DPIT301.SAHH, SAH := HMI_DPIT301.SAH, SAL := HMI_DPIT301.SAL, SALL := HMI_DPIT301.SALL, Simulation := HMI_DPIT301.Sim, RIO_Hty := AI_DPIT_301_DPRESS_HTY, WRIO_Hty := W_AI_DPIT_301_DPRESS_HTY, HMI := HMI_DPIT301, Pv := HMI_DPIT301.Pv, Sim_PV := HMI_DPIT301.Sim_PV);
   HMI_PSH301.Alarm := PSH301_FB.Status;
   HMI_DPSH301.Alarm := DPSH301_FB.Status;
   HMI_DPIT301.Wifi_Enb := DPIT301_FB.Wifi_Enb;
   HMI_DPIT301.Hty := DPIT301_FB.Hty;
   HMI_DPIT301.AHH := DPIT301_FB.AHH;
   HMI_DPIT301.AH := DPIT301_FB.AH;
   HMI_DPIT301.ALL := DPIT301_FB.ALL;
   HMI_DPIT301.AL := DPIT301_FB.AL;
   MV301_FB : MV_FBD(Auto := HMI_MV301.Auto, AutoInp := _MV301_AutoInp, ZSO := DI_MV_301_ZSO, Open_TM := 10, ZSC := DI_MV_301_ZSC, Close_TM := 10, Cmd := HMI_MV301.Cmd, HMI := HMI_MV301);
   MV302_FB : MV_FBD(Auto := HMI_MV302.Auto, AutoInp := _MV302_AutoInp, ZSO := DI_MV_302_ZSO, Open_TM := 10, ZSC := DI_MV_302_ZSC, Close_TM := 10, Cmd := HMI_MV302.Cmd, HMI := HMI_MV302);
   MV303_FB : MV_FBD(Auto := HMI_MV303.Auto, AutoInp := _MV303_AutoInp, ZSO := DI_MV_303_ZSO, Open_TM := 10, ZSC := DI_MV_303_ZSC, Close_TM := 10, Cmd := HMI_MV303.Cmd, HMI := HMI_MV303);
   MV304_FB : MV_FBD(Auto := HMI_MV304.Auto, AutoInp := _MV304_AutoInp, ZSO := DI_MV_304_ZSO, Open_TM := 10, ZSC := DI_MV_304_ZSC, Close_TM := 10, Cmd := HMI_MV304.Cmd, HMI := HMI_MV304);
   DO_MV_301_CLOSE := MV301_FB.Cmd_Close;
   DO_MV_302_CLOSE := MV302_FB.Cmd_Close;
   DO_MV_301_OPEN := MV301_FB.Cmd_Open;
   DO_MV_302_OPEN := MV302_FB.Cmd_Open;
   HMI_MV301.FTO := MV301_FB.FTO;
   HMI_MV302.FTO := MV302_FB.FTO;
   HMI_MV301.FTC := MV301_FB.FTC;
   HMI_MV302.FTC := MV302_FB.FTC;
   DO_MV_303_CLOSE := MV303_FB.Cmd_Close;
   DO_MV_303_OPEN := MV303_FB.Cmd_Open;
   DO_MV_304_OPEN := MV304_FB.Cmd_Open;
   HMI_MV304.FTC := MV304_FB.FTC;
   HMI_MV303.FTO := MV303_FB.FTO;
   HMI_MV303.FTC := MV303_FB.FTC;
   DO_MV_304_CLOSE := MV304_FB.Cmd_Close;
   HMI_MV304.FTO := MV304_FB.FTO;
END_ROUTINE

ROUTINE Validate_Input   (* structured text *)
// Validating Input by Historical values
   (*SECOND PULSE*)
   TON1.PRE	:=1000;
   TON1.TimerEnable	:=1;
   TONR(TON1 );
   R_TRIG1.InputBit :=TON1.DN ;
   OSRI( R_TRIG1);
   _SEC_P3  := R_TRIG1.OutputBit;
   TON1.Reset := _SEC_P3;
   
   IF  _SEC_P      THEN
   	SEC_TEST:=SEC_TEST+1;
       _SEC_P_2 := 1;         (* we made it *)
   END_IF;
   
   IF  SEC_TEST = 60   THEN
   	_MIN_P  := 1;
   	SEC_TEST:=0;
   END_IF;
   
   
   
   
   IF HMI_PLANT.START OR HMI_PLANT.STOP   THEN
   	LIT_STATE:=0;
   END_IF;
   
   
   
   //CASE STATEMENT CHECKS THE LIT301 WITH RESPECT TO FIT201 AND FIT301
   CASE LIT_STATE OF
   
   	0:(*  dummy state *)
   		LIT_301_Le_PRV		:= HMI_LIT301.Pv ;
   		LIT_301_Ls_PRV		:= HMI_LIT301.Pv ;
   		LIT_STATE		:= 1;
   		ERROR_P3_Le := 0;
   		ERROR_P3_Ls := 0;
   		Ls_Error_Occured := 0;
   		Le_Error_Occured := 0;
   
   	1:(* *)
   
   		LIT_SEC_SP 		:= 5;
   		LIT_SEC			:= 0;
   		LIT_STATE		:= 2;
   
   	2:
           IF _SEC_P_2 THEN
   		(*LIT_SEC := LIT_SEC+1;
   				_SEC_P_2 :=0;
   			IF LIT_SEC > LIT_SEC_SP THEN
   				LIT_STATE:=3;
   				LIT_SEC:=0;
   			END_IF;*)
   			LIT_STATE:=4;
   		    _SEC_P_2 :=0;
   		END_IF;
   		LIT_SEC := LIT_SEC+1;
   	3:
   		IF _SEC_P_2 THEN
   			LIT_STATE:=4;     (*  NOT USING THIS CODE, JUMPING TO NEXT STATE *)
   		    _SEC_P_2 :=0;
   		END_IF;
   	4:
   		 LIT_301_MODEL_Ls 	:=  LIT_301_Ls_PRV + ((HMI_FIT201.Pv - HMI_FIT301.Pv) * 0.186428);
   		 LIT_301_Ls_PRV		:= 	HMI_LIT301.Pv ; (* Assign Updated sensor's value *)
    		 ERROR_P3_Ls := ABS(LIT_301_MODEL_Ls - HMI_LIT301.Pv);
   
   		 Error_list[count] := ERROR_P3_Ls;
   		 IF first THEN
   		    avg := ( Error_list[9]+Error_list[8]+Error_list[7]+Error_list[6]+Error_list[5]+Error_list[4]+Error_list[3]+Error_list[2]+Error_list[1]+ Error_list[0] ) /10;
   		END_IF;
   		count := count + 1;
   		IF count > 9 THEN
   			count := 0;
   			first := 1;
   		END_IF;
   
   		 //LIT_301_MODEL_Le 	:=  LIT_301_Le_PRV + ((HMI_FIT201.Pv - HMI_FIT301.Pv+0.003) * 0.1864);
   		 //LIT_301_Le_PRV		:= 	LIT_301_MODEL_Le ; (* Assign Updated model value *)
   		 //ERROR_P3_Le := ABS(LIT_301_MODEL_Le - HMI_LIT301.Pv);
            LIT_SEC			:= 0;
   		 IF ERROR_P3_Ls > 4.00 THEN
   			LIT_STATE			:=	5;
   		// ELSIF ERROR_P3_Le > 20.00 THEN
   		//	LIT_STATE			:=	6;
   		 ELSE
   		 	LIT_STATE			:=	2;
   		 END_IF;
   	5:   Ls_Error_Occured := 1; LIT_STATE			:=	2;
   	6:   Le_Error_Occured := 1; LIT_STATE			:=	2;
   
   ELSE
   	LIT_STATE:=1;
   END_CASE;
   
   
   //BACKWARD CHECKING
   (* LIT301 LOW THEN MV201 SHOULD OPEN AND P101 SHOULD BE ON *)
   (* LIT301 HIgh HIGH THEN MV201 SHOULD BE CLOSE AND P101 SHOULD BE OFF *)
   
   
   (* LIT301 LOW THEN MV201 SHOULD OPEN AND P101 SHOULD BE ON *)
   IF HMI_LIT301.AL THEN
   	IF _MIN_P THEN
     //TIME
   		IF HMI_MV201.Status <> 2  THEN
   			ATTACK := 1;
   		END_IF;
   		IF HMI_P101.Status <> 2 THEN
   			ATTACK :=1;
   		END_IF;
   	END_IF;
   END_IF;
   
   
   
   (* LIT301 HIgh THEN MV201 SHOULD BE CLOSE AND P101 SHOULD BE OFF *)
   
   IF HMI_LIT301.AH THEN
   	IF _MIN_P THEN
   //TIME
   		IF HMI_MV201.Status <> 1  THEN
   			ATTACK := 1;
   		END_IF;
   		IF HMI_P101.Status <> 1 THEN
   			ATTACK :=1;
   		END_IF;
   	END_IF;
   END_IF;
   
   
   
   
   
   //FORWARD CHECKING
   
   (* LIT301 LOW LOW THEN PUMP P301 SHOULD BE STOP   *)
   IF HMI_LIT301.ALL THEN
   	IF _MIN_P THEN
   //TIME
   		IF HMI_P301.Status <> 2 THEN
   			ATTACK :=1;
   		END_IF;
   	END_IF;
   END_IF;
   
   
   
   (* PUMP P301 ON THEN FIT301 SHOULD HAVE SOME VALUE*)
   
   IF HMI_P301.Status = 2 THEN
   	IF _MIN_P THEN
   //TIME
   		IF HMI_FIT301.Pv < 1 THEN
   			ATTACK :=1;
   		END_IF;
   	END_IF;
   END_IF;
   
   
   (* HMI_DPIT301.AH MEANS DPIT301 HIGH PUMP P301 SHOULD STOP   *)
   IF HMI_DPIT301.AH THEN
   	IF _MIN_P THEN
   //TIME
   		IF HMI_P301.Status = 2 THEN
   			ATTACK :=1;
   		END_IF;
   	END_IF;
   END_IF;
   
   (* HOW TO ADD CONDITIONS FROM STAGE 4 BY OVERCOMING THE BACKWASH TIME: use MV302 *)
   
   
   (*   WHEN LIT401 LOW PUMP P301 SHOULD RUN OR MV302 SHOULD BE OPEN*)
   
   (*IF HMI_LIT401.AL THEN
   	IF _MIN_P THEN
   //TIME
   		IF HMI_P301.Status = 1 AND HMI_MV302.Status = 1 THEN
   			ATTACK :=1;
   		END_IF;
   	END_IF;
   END_IF; *)
   
   
   (*   WHEN LIT401 LOW PUMP P301 SHOULD RUN OR MV302 SHOULD BE OPEN*)
   IF HMI_LIT401.AL THEN
   	IF _MIN_P THEN
   		IF HMI_P301.Status = 1  AND HMI_MV301.Status = 1 AND HMI_MV302.Status = 1 AND HMI_MV303.Status = 1 AND HMI_MV304.Status = 1 THEN
   			ATTACK :=1;
   		END_IF;
   	END_IF;
   END_IF;
   
   
   (*  LIT401 HIGH PUMP P301 SHOULD BE STOP  *)
   IF HMI_LIT401.AH THEN
   	IF _MIN_P THEN
   	//TIME
   		IF HMI_P301.Status = 2 THEN
   			ATTACK :=1;
   		END_IF;
   	END_IF;
   END_IF;
   
   
   
END_ROUTINE
END_PROGRAM
